LIN {X 0,Y 220.373,Z 1009.836,A -85,B 0,C 180,E1 18253.847,E2 18253.847} C_VEL
LIN {X 0,Y 219.138,Z 1016.029,A -85,B 0,C 180,E1 18268.015,E2 18268.015} C_VEL
LIN {X 0,Y 219.565,Z 1013.034,A -85,B 0,C 180,E1 18281.966,E2 18281.966} C_VEL
LIN {X 0,Y 227.617,Z 997.179,A -85,B 0,C 180,E1 18298.905,E2 18298.905} C_VEL
LIN {X 0,Y 250.356,Z 965.181,A -85,B 0,C 180,E1 18314.989,E2 18314.989} C_VEL
LIN {X 0,Y 283.389,Z 919.125,A -85,B 0,C 180,E1 18326.696,E2 18326.696} C_VEL
LIN {X 0,Y 317.274,Z 862.724,A -85,B 0,C 180,E1 18334.047,E2 18334.047} C_VEL
LIN {X 0,Y 322.512,Z 850.682,A -85,B 0,C 180,E1 18335.556,E2 18335.556} C_VEL
LIN {X 0,Y 322.481,Z 836.456,A -85,B 0,C 180,E1 18342.214,E2 18342.214} C_VEL
LIN {X 0,Y 322.225,Z 833.773,A -85,B 0,C 180,E1 18347.787,E2 18347.787} C_VEL
LIN {X 0,Y 321.726,Z 841.185,A -85,B 0,C 180,E1 18353.928,E2 18353.928} C_VEL
LIN {X 0,Y 319.566,Z 854.404,A -85,B 0,C 180,E1 18358.488,E2 18358.488} C_VEL
LIN {X 0,Y 300.592,Z 887.455,A -85,B 0,C 180,E1 18362.382,E2 18362.382} C_VEL
LIN {X 0,Y 279.885,Z 912.877,A -85,B 0,C 180,E1 18365.051,E2 18365.051} C_VEL
LIN {X 0,Y 246.942,Z 954.001,A -85,B 0,C 180,E1 18376.073,E2 18376.073} C_VEL
LIN {X 0,Y 222.563,Z 982.704,A -85,B 0,C 180,E1 18391.535,E2 18391.535} C_VEL
LIN {X 0,Y 212.303,Z 997.242,A -85,B 0,C 180,E1 18408.658,E2 18408.658} C_VEL
LIN {X 0,Y 209.744,Z 999.849,A -85,B 0,C 180,E1 18424.769,E2 18424.769} C_VEL
LIN {X 0,Y 214.305,Z 991.756,A -85,B 0,C 180,E1 18441.286,E2 18441.286} C_VEL
LIN {X 0,Y 227.941,Z 970.708,A -85,B 0,C 180,E1 18457.653,E2 18457.653} C_VEL
LIN {X 0,Y 253.573,Z 935.333,A -85,B 0,C 180,E1 18471.372,E2 18471.372} C_VEL
LIN {X 0,Y 285.146,Z 885.566,A -85,B 0,C 180,E1 18481.26,E2 18481.26} C_VEL
LIN {X 0,Y 302.468,Z 850.539,A -85,B 0,C 180,E1 18485.569,E2 18485.569} C_VEL
LIN {X 0,Y 296.04,Z 820.813,A -85,B 0,C 180,E1 18495.646,E2 18495.646} C_VEL
LIN {X 0,Y 288.186,Z 798.555,A -85,B 0,C 180,E1 18507.321,E2 18507.321} C_VEL
LIN {X 0,Y 283.718,Z 785.2,A -85,B 0,C 180,E1 18521.323,E2 18521.323} C_VEL
LIN {X 0,Y 285.026,Z 786.25,A -85,B 0,C 180,E1 18533.316,E2 18533.316} C_VEL
LIN {X 0,Y 290.912,Z 799.543,A -85,B 0,C 180,E1 18545.216,E2 18545.216} C_VEL
LIN {X 0,Y 300.284,Z 824.928,A -85,B 0,C 180,E1 18556.867,E2 18556.867} C_VEL
LIN {X 0,Y 306.026,Z 852.939,A -85,B 0,C 180,E1 18565.183,E2 18565.183} C_VEL
LIN {X 0,Y 276.942,Z 909.709,A -85,B 0,C 180,E1 18571.855,E2 18571.855} C_VEL
LIN {X 0,Y 245.558,Z 958.022,A -85,B 0,C 180,E1 18582.734,E2 18582.734} C_VEL
LIN {X 0,Y 221.833,Z 992.283,A -85,B 0,C 180,E1 18597.981,E2 18597.981} C_VEL
LIN {X 0,Y 212.147,Z 1010.601,A -85,B 0,C 180,E1 18614.772,E2 18614.772} C_VEL
LIN {X 0,Y 211.129,Z 1015.72,A -85,B 0,C 180,E1 18627.939,E2 18627.939} C_VEL
LIN {X 0,Y 211.636,Z 1012.762,A -85,B 0,C 180,E1 18642.422,E2 18642.422} C_VEL
LIN {X 0,Y 220.353,Z 997.009,A -85,B 0,C 180,E1 18659.954,E2 18659.954} C_VEL
LIN {X 0,Y 244.372,Z 965.392,A -85,B 0,C 180,E1 18676.307,E2 18676.307} C_VEL
LIN {X 0,Y 278.886,Z 919.71,A -85,B 0,C 180,E1 18688.066,E2 18688.066} C_VEL
LIN {X 0,Y 313.812,Z 864.077,A -85,B 0,C 180,E1 18695.333,E2 18695.333} C_VEL
LIN {X 0,Y 317.905,Z 855.344,A -85,B 0,C 180,E1 18696.473,E2 18696.473} C_VEL
LIN {X 0,Y 318.346,Z 842.413,A -85,B 0,C 180,E1 18703.405,E2 18703.405} C_VEL
LIN {X 0,Y 318.197,Z 842.388,A -85,B 0,C 180,E1 18710.413,E2 18710.413} C_VEL
LIN {X 0,Y 315.699,Z 857.128,A -85,B 0,C 180,E1 18717.308,E2 18717.308} C_VEL
LIN {X 0,Y 281.373,Z 910.889,A -85,B 0,C 180,E1 18724.66,E2 18724.66} C_VEL
LIN {X 0,Y 279.885,Z 912.877,A -85,B 0,C 180,E1 18725.051,E2 18725.051} C_VEL
LIN {X 0,Y 258.115,Z 935.593,A -85,B 0,C 180,E1 18728.56,E2 18728.56} C_VEL
LIN {X 0,Y 226.791,Z 970.834,A -85,B 0,C 180,E1 18742.183,E2 18742.183} C_VEL
LIN {X 0,Y 207.855,Z 992.665,A -85,B 0,C 180,E1 18759.95,E2 18759.95} C_VEL
LIN {X 0,Y 202.185,Z 999.999,A -85,B 0,C 180,E1 18775.741,E2 18775.741} C_VEL
LIN {X 0,Y 203.21,Z 997.796,A -85,B 0,C 180,E1 18792.62,E2 18792.62} C_VEL
LIN {X 0,Y 211.901,Z 983.961,A -85,B 0,C 180,E1 18809.984,E2 18809.984} C_VEL
LIN {X 0,Y 234.192,Z 954.323,A -85,B 0,C 180,E1 18826.47,E2 18826.47} C_VEL
LIN {X 0,Y 263.333,Z 913.447,A -85,B 0,C 180,E1 18837.921,E2 18837.921} C_VEL
LIN {X 0,Y 293.981,Z 860.719,A -85,B 0,C 180,E1 18845.731,E2 18845.731} C_VEL
LIN {X 0,Y 296.609,Z 852.495,A -85,B 0,C 180,E1 18847.039,E2 18847.039} C_VEL
LIN {X 0,Y 290.792,Z 824.048,A -85,B 0,C 180,E1 18857.396,E2 18857.396} C_VEL
LIN {X 0,Y 283.733,Z 803.211,A -85,B 0,C 180,E1 18869.449,E2 18869.449} C_VEL
LIN {X 0,Y 280.825,Z 792.085,A -85,B 0,C 180,E1 18882.693,E2 18882.693} C_VEL
LIN {X 0,Y 282.263,Z 794.533,A -85,B 0,C 180,E1 18894.079,E2 18894.079} C_VEL
LIN {X 0,Y 287.729,Z 807.162,A -85,B 0,C 180,E1 18905.273,E2 18905.273} C_VEL
LIN {X 0,Y 296.059,Z 832.031,A -85,B 0,C 180,E1 18916.731,E2 18916.731} C_VEL
LIN {X 0,Y 300.062,Z 857.017,A -85,B 0,C 180,E1 18924.226,E2 18924.226} C_VEL
LIN {X 0,Y 270.046,Z 912.728,A -85,B 0,C 180,E1 18931.016,E2 18931.016} C_VEL
LIN {X 0,Y 238.555,Z 959.182,A -85,B 0,C 180,E1 18941.859,E2 18941.859} C_VEL
LIN {X 0,Y 214.827,Z 991.776,A -85,B 0,C 180,E1 18956.805,E2 18956.805} C_VEL
LIN {X 0,Y 204.65,Z 1009.197,A -85,B 0,C 180,E1 18972.744,E2 18972.744} C_VEL
LIN {X 0,Y 203.132,Z 1015.411,A -85,B 0,C 180,E1 18987.858,E2 18987.858} C_VEL
LIN {X 0,Y 203.701,Z 1012.495,A -85,B 0,C 180,E1 19002.914,E2 19002.914} C_VEL
LIN {X 0,Y 213.159,Z 996.874,A -85,B 0,C 180,E1 19021.055,E2 19021.055} C_VEL
LIN {X 0,Y 239.014,Z 965.037,A -85,B 0,C 180,E1 19037.919,E2 19037.919} C_VEL
LIN {X 0,Y 275.385,Z 919.278,A -85,B 0,C 180,E1 19049.672,E2 19049.672} C_VEL
LIN {X 0,Y 311.753,Z 863.373,A -85,B 0,C 180,E1 19056.851,E2 19056.851} C_VEL
LIN {X 0,Y 313.841,Z 854.831,A -85,B 0,C 180,E1 19059.622,E2 19059.622} C_VEL
LIN {X 0,Y 314.074,Z 848.409,A -85,B 0,C 180,E1 19064.613,E2 19064.613} C_VEL
LIN {X 0,Y 313.639,Z 850.576,A -85,B 0,C 180,E1 19071.382,E2 19071.382} C_VEL
LIN {X 0,Y 310.047,Z 863.365,A -85,B 0,C 180,E1 19076.454,E2 19076.454} C_VEL
LIN {X 0,Y 273.828,Z 916.35,A -85,B 0,C 180,E1 19084.114,E2 19084.114} C_VEL
LIN {X 0,Y 258.115,Z 935.593,A -85,B 0,C 180,E1 19088.56,E2 19088.56} C_VEL
LIN {X 0,Y 236.075,Z 955.304,A -85,B 0,C 180,E1 19093.128,E2 19093.128} C_VEL
LIN {X 0,Y 208.191,Z 984.166,A -85,B 0,C 180,E1 19109.592,E2 19109.592} C_VEL
LIN {X 0,Y 196.123,Z 998.481,A -85,B 0,C 180,E1 19128.875,E2 19128.875} C_VEL
LIN {X 0,Y 193.672,Z 1000.479,A -85,B 0,C 180,E1 19144.472,E2 19144.472} C_VEL
LIN {X 0,Y 197.918,Z 993.812,A -85,B 0,C 180,E1 19160.495,E2 19160.495} C_VEL
LIN {X 0,Y 211.983,Z 974.227,A -85,B 0,C 180,E1 19178.233,E2 19178.233} C_VEL
LIN {X 0,Y 239.645,Z 939.396,A -85,B 0,C 180,E1 19193.058,E2 19193.058} C_VEL
LIN {X 0,Y 272.06,Z 892.564,A -85,B 0,C 180,E1 19203.038,E2 19203.038} C_VEL
LIN {X 0,Y 291.019,Z 856.591,A -85,B 0,C 180,E1 19207.905,E2 19207.905} C_VEL
LIN {X 0,Y 285.972,Z 828.948,A -85,B 0,C 180,E1 19218.435,E2 19218.435} C_VEL
LIN {X 0,Y 280.548,Z 811.013,A -85,B 0,C 180,E1 19229.064,E2 19229.064} C_VEL
LIN {X 0,Y 277.851,Z 799.48,A -85,B 0,C 180,E1 19242.909,E2 19242.909} C_VEL
LIN {X 0,Y 279.25,Z 801.961,A -85,B 0,C 180,E1 19254.015,E2 19254.015} C_VEL
LIN {X 0,Y 284.31,Z 814.699,A -85,B 0,C 180,E1 19265.337,E2 19265.337} C_VEL
LIN {X 0,Y 291.619,Z 838.957,A -85,B 0,C 180,E1 19276.605,E2 19276.605} C_VEL
LIN {X 0,Y 294.508,Z 860.273,A -85,B 0,C 180,E1 19283.162,E2 19283.162} C_VEL
LIN {X 0,Y 263.242,Z 915.713,A -85,B 0,C 180,E1 19290.144,E2 19290.144} C_VEL
LIN {X 0,Y 231.356,Z 960.576,A -85,B 0,C 180,E1 19301.03,E2 19301.03} C_VEL
LIN {X 0,Y 206.727,Z 992.867,A -85,B 0,C 180,E1 19316.592,E2 19316.592} C_VEL
LIN {X 0,Y 196.236,Z 1010.295,A -85,B 0,C 180,E1 19334.295,E2 19334.295} C_VEL
LIN {X 0,Y 195.12,Z 1015.1,A -85,B 0,C 180,E1 19347.77,E2 19347.77} C_VEL
LIN {X 0,Y 195.48,Z 1013.18,A -85,B 0,C 180,E1 19361.19,E2 19361.19} C_VEL
LIN {X 0,Y 204.534,Z 998.649,A -85,B 0,C 180,E1 19380.621,E2 19380.621} C_VEL
LIN {X 0,Y 230.077,Z 968.974,A -85,B 0,C 180,E1 19397.905,E2 19397.905} C_VEL
LIN {X 0,Y 266.944,Z 925.543,A -85,B 0,C 180,E1 19410.107,E2 19410.107} C_VEL
LIN {X 0,Y 306.085,Z 869.504,A -85,B 0,C 180,E1 19417.76,E2 19417.76} C_VEL
LIN {X 0,Y 309.026,Z 862.483,A -85,B 0,C 180,E1 19419.29,E2 19419.29} C_VEL
LIN {X 0,Y 309.799,Z 855.412,A -85,B 0,C 180,E1 19424.396,E2 19424.396} C_VEL
LIN {X 0,Y 309.551,Z 855.889,A -85,B 0,C 180,E1 19430.143,E2 19430.143} C_VEL
LIN {X 0,Y 306.388,Z 866.253,A -85,B 0,C 180,E1 19435.226,E2 19435.226} C_VEL
LIN {X 0,Y 268.378,Z 919.194,A -85,B 0,C 180,E1 19442.994,E2 19442.994} C_VEL
LIN {X 0,Y 236.075,Z 955.304,A -85,B 0,C 180,E1 19453.128,E2 19453.128} C_VEL
LIN {X 0,Y 214.987,Z 971.635,A -85,B 0,C 180,E1 19459.091,E2 19459.091} C_VEL
LIN {X 0,Y 192.996,Z 993.395,A -85,B 0,C 180,E1 19477.924,E2 19477.924} C_VEL
LIN {X 0,Y 186.819,Z 1000.134,A -85,B 0,C 180,E1 19492.466,E2 19492.466} C_VEL
LIN {X 0,Y 186.364,Z 999.741,A -85,B 0,C 180,E1 19509.501,E2 19509.501} C_VEL
LIN {X 0,Y 192.215,Z 990.787,A -85,B 0,C 180,E1 19525.532,E2 19525.532} C_VEL
LIN {X 0,Y 211.117,Z 967.464,A -85,B 0,C 180,E1 19543.533,E2 19543.533} C_VEL
LIN {X 0,Y 242.514,Z 928.84,A -85,B 0,C 180,E1 19557.485,E2 19557.485} C_VEL
LIN {X 0,Y 276.181,Z 878.662,A -85,B 0,C 180,E1 19566.452,E2 19566.452} C_VEL
LIN {X 0,Y 285.512,Z 860.953,A -85,B 0,C 180,E1 19568.708,E2 19568.708} C_VEL
LIN {X 0,Y 281.244,Z 834.112,A -85,B 0,C 180,E1 19579.384,E2 19579.384} C_VEL
LIN {X 0,Y 276.401,Z 816.717,A -85,B 0,C 180,E1 19590.458,E2 19590.458} C_VEL
LIN {X 0,Y 274.593,Z 806.641,A -85,B 0,C 180,E1 19605.281,E2 19605.281} C_VEL
LIN {X 0,Y 276.326,Z 810.262,A -85,B 0,C 180,E1 19615.255,E2 19615.255} C_VEL
LIN {X 0,Y 281.536,Z 824.755,A -85,B 0,C 180,E1 19626.942,E2 19626.942} C_VEL
LIN {X 0,Y 287.874,Z 850.107,A -85,B 0,C 180,E1 19638.014,E2 19638.014} C_VEL
LIN {X 0,Y 288.564,Z 864.213,A -85,B 0,C 180,E1 19642.155,E2 19642.155} C_VEL
LIN {X 0,Y 256.518,Z 918.691,A -85,B 0,C 180,E1 19649.236,E2 19649.236} C_VEL
LIN {X 0,Y 222.348,Z 964.299,A -85,B 0,C 180,E1 19660.992,E2 19660.992} C_VEL
LIN {X 0,Y 197.99,Z 994.596,A -85,B 0,C 180,E1 19676.98,E2 19676.98} C_VEL
LIN {X 0,Y 188.368,Z 1009.917,A -85,B 0,C 180,E1 19693.621,E2 19693.621} C_VEL
LIN {X 0,Y 187.121,Z 1014.79,A -85,B 0,C 180,E1 19707.675,E2 19707.675} C_VEL
LIN {X 0,Y 187.765,Z 1012.235,A -85,B 0,C 180,E1 19723.373,E2 19723.373} C_VEL
LIN {X 0,Y 198.68,Z 997.07,A -85,B 0,C 180,E1 19743.168,E2 19743.168} C_VEL
LIN {X 0,Y 228.668,Z 964.789,A -85,B 0,C 180,E1 19761.194,E2 19761.194} C_VEL
LIN {X 0,Y 268.282,Z 919.662,A -85,B 0,C 180,E1 19772.816,E2 19772.816} C_VEL
LIN {X 0,Y 304.265,Z 868.851,A -85,B 0,C 180,E1 19779.581,E2 19779.581} C_VEL
LIN {X 0,Y 305.188,Z 861.542,A -85,B 0,C 180,E1 19785.849,E2 19785.849} C_VEL
LIN {X 0,Y 304.29,Z 864.506,A -85,B 0,C 180,E1 19791.418,E2 19791.418} C_VEL
LIN {X 0,Y 300.81,Z 872.287,A -85,B 0,C 180,E1 19794.309,E2 19794.309} C_VEL
LIN {X 0,Y 261.63,Z 923.52,A -85,B 0,C 180,E1 19802.173,E2 19802.173} C_VEL
LIN {X 0,Y 224.173,Z 962.683,A -85,B 0,C 180,E1 19814.39,E2 19814.39} C_VEL
LIN {X 0,Y 214.987,Z 971.635,A -85,B 0,C 180,E1 19819.091,E2 19819.091} C_VEL
LIN {X 0,Y 195.178,Z 984.685,A -85,B 0,C 180,E1 19826.484,E2 19826.484} C_VEL
LIN {X 0,Y 181.146,Z 998.421,A -85,B 0,C 180,E1 19845.432,E2 19845.432} C_VEL
LIN {X 0,Y 177.585,Z 1001.129,A -85,B 0,C 180,E1 19863.839,E2 19863.839} C_VEL
LIN {X 0,Y 181.808,Z 995.317,A -85,B 0,C 180,E1 19880.391,E2 19880.391} C_VEL
LIN {X 0,Y 197.338,Z 975.911,A -85,B 0,C 180,E1 19899.965,E2 19899.965} C_VEL
LIN {X 0,Y 226.305,Z 942.826,A -85,B 0,C 180,E1 19915.118,E2 19915.118} C_VEL
LIN {X 0,Y 261.524,Z 895.866,A -85,B 0,C 180,E1 19925.53,E2 19925.53} C_VEL
LIN {X 0,Y 279.861,Z 863.813,A -85,B 0,C 180,E1 19930.039,E2 19930.039} C_VEL
LIN {X 0,Y 276.366,Z 838.353,A -85,B 0,C 180,E1 19940.829,E2 19940.829} C_VEL
LIN {X 0,Y 272.298,Z 822.591,A -85,B 0,C 180,E1 19951.71,E2 19951.71} C_VEL
LIN {X 0,Y 271.325,Z 813.923,A -85,B 0,C 180,E1 19965.405,E2 19965.405} C_VEL
LIN {X 0,Y 272.968,Z 817.502,A -85,B 0,C 180,E1 19975.196,E2 19975.196} C_VEL
LIN {X 0,Y 277.749,Z 832.214,A -85,B 0,C 180,E1 19987.038,E2 19987.038} C_VEL
LIN {X 0,Y 283.068,Z 857.304,A -85,B 0,C 180,E1 19998.07,E2 19998.07} C_VEL
LIN {X 0,Y 282.572,Z 868.253,A -85,B 0,C 180,E1 20001.117,E2 20001.117} C_VEL
LIN {X 0,Y 249.814,Z 921.374,A -85,B 0,C 180,E1 20008.253,E2 20008.253} C_VEL
LIN {X 0,Y 215.743,Z 964.986,A -85,B 0,C 180,E1 20019.832,E2 20019.832} C_VEL
LIN {X 0,Y 189.597,Z 995.901,A -85,B 0,C 180,E1 20037.098,E2 20037.098} C_VEL
LIN {X 0,Y 179.879,Z 1011.008,A -85,B 0,C 180,E1 20055.766,E2 20055.766} C_VEL
LIN {X 0,Y 179.299,Z 1014.62,A -85,B 0,C 180,E1 20072.424,E2 20072.424} C_VEL
LIN {X 0,Y 182.377,Z 1007.844,A -85,B 0,C 180,E1 20091.989,E2 20091.989} C_VEL
LIN {X 0,Y 201.967,Z 986.21,A -85,B 0,C 180,E1 20112.551,E2 20112.551} C_VEL
LIN {X 0,Y 238.666,Z 949.421,A -85,B 0,C 180,E1 20127.929,E2 20127.929} C_VEL
LIN {X 0,Y 280.238,Z 901.075,A -85,B 0,C 180,E1 20137.335,E2 20137.335} C_VEL
LIN {X 0,Y 299.708,Z 873.201,A -85,B 0,C 180,E1 20140.812,E2 20140.812} C_VEL
LIN {X 0,Y 300.756,Z 867.825,A -85,B 0,C 180,E1 20146.901,E2 20146.901} C_VEL
LIN {X 0,Y 298.717,Z 872.659,A -85,B 0,C 180,E1 20152.131,E2 20152.131} C_VEL
LIN {X 0,Y 293.823,Z 880.361,A -85,B 0,C 180,E1 20153.608,E2 20153.608} C_VEL
LIN {X 0,Y 253.158,Z 929.782,A -85,B 0,C 180,E1 20161.74,E2 20161.74} C_VEL
LIN {X 0,Y 214.089,Z 967.716,A -85,B 0,C 180,E1 20174.957,E2 20174.957} C_VEL
LIN {X 0,Y 195.178,Z 984.685,A -85,B 0,C 180,E1 20186.484,E2 20186.484} C_VEL
LIN {X 0,Y 178.309,Z 994.199,A -85,B 0,C 180,E1 20195.666,E2 20195.666} C_VEL
LIN {X 0,Y 170.224,Z 1001.371,A -85,B 0,C 180,E1 20214.587,E2 20214.587} C_VEL
LIN {X 0,Y 171.766,Z 998.594,A -85,B 0,C 180,E1 20235.07,E2 20235.07} C_VEL
LIN {X 0,Y 183.906,Z 983.75,A -85,B 0,C 180,E1 20255.332,E2 20255.332} C_VEL
LIN {X 0,Y 211.438,Z 954.189,A -85,B 0,C 180,E1 20272.694,E2 20272.694} C_VEL
LIN {X 0,Y 247.11,Z 910.522,A -85,B 0,C 180,E1 20284.617,E2 20284.617} C_VEL
LIN {X 0,Y 274.285,Z 868.117,A -85,B 0,C 180,E1 20290.87,E2 20290.87} C_VEL
LIN {X 0,Y 271.715,Z 844.511,A -85,B 0,C 180,E1 20301.256,E2 20301.256} C_VEL
LIN {X 0,Y 268.173,Z 827.819,A -85,B 0,C 180,E1 20313.613,E2 20313.613} C_VEL
LIN {X 0,Y 267.755,Z 821.155,A -85,B 0,C 180,E1 20325.206,E2 20325.206} C_VEL
LIN {X 0,Y 269.313,Z 824.6,A -85,B 0,C 180,E1 20335.131,E2 20335.131} C_VEL
LIN {X 0,Y 273.617,Z 839.556,A -85,B 0,C 180,E1 20347.144,E2 20347.144} C_VEL
LIN {X 0,Y 277.981,Z 863.95,A -85,B 0,C 180,E1 20357.976,E2 20357.976} C_VEL
LIN {X 0,Y 277.354,Z 870.945,A -85,B 0,C 180,E1 20359.909,E2 20359.909} C_VEL
LIN {X 0,Y 242.904,Z 924.412,A -85,B 0,C 180,E1 20367.306,E2 20367.306} C_VEL
LIN {X 0,Y 208.121,Z 966.819,A -85,B 0,C 180,E1 20379.087,E2 20379.087} C_VEL
LIN {X 0,Y 181.35,Z 996.976,A -85,B 0,C 180,E1 20397.047,E2 20397.047} C_VEL
LIN {X 0,Y 171.656,Z 1011.578,A -85,B 0,C 180,E1 20417.23,E2 20417.23} C_VEL
LIN {X 0,Y 171.299,Z 1014.33,A -85,B 0,C 180,E1 20432.538,E2 20432.538} C_VEL
LIN {X 0,Y 174.747,Z 1007.653,A -85,B 0,C 180,E1 20453.003,E2 20453.003} C_VEL
LIN {X 0,Y 195.931,Z 986.211,A -85,B 0,C 180,E1 20474.193,E2 20474.193} C_VEL
LIN {X 0,Y 234.661,Z 949.6,A -85,B 0,C 180,E1 20489.701,E2 20489.701} C_VEL
LIN {X 0,Y 277.708,Z 901.724,A -85,B 0,C 180,E1 20498.913,E2 20498.913} C_VEL
LIN {X 0,Y 295.194,Z 877.852,A -85,B 0,C 180,E1 20502.003,E2 20502.003} C_VEL
LIN {X 0,Y 295.893,Z 874.332,A -85,B 0,C 180,E1 20506.681,E2 20506.681} C_VEL
LIN {X 0,Y 294.382,Z 877.613,A -85,B 0,C 180,E1 20511.127,E2 20511.127} C_VEL
LIN {X 0,Y 285.888,Z 889.367,A -85,B 0,C 180,E1 20513.015,E2 20513.015} C_VEL
LIN {X 0,Y 242.563,Z 937.712,A -85,B 0,C 180,E1 20521.816,E2 20521.816} C_VEL
LIN {X 0,Y 203.626,Z 972.739,A -85,B 0,C 180,E1 20535.745,E2 20535.745} C_VEL
LIN {X 0,Y 178.309,Z 994.199,A -85,B 0,C 180,E1 20555.666,E2 20555.666} C_VEL
LIN {X 0,Y 164.556,Z 1000.038,A -85,B 0,C 180,E1 20566.474,E2 20566.474} C_VEL
LIN {X 0,Y 161.52,Z 1001.635,A -85,B 0,C 180,E1 20584.989,E2 20584.989} C_VEL
LIN {X 0,Y 167.196,Z 994.523,A -85,B 0,C 180,E1 20604.065,E2 20604.065} C_VEL
LIN {X 0,Y 185.998,Z 974.459,A -85,B 0,C 180,E1 20624.17,E2 20624.17} C_VEL
LIN {X 0,Y 219.864,Z 938.759,A -85,B 0,C 180,E1 20639.736,E2 20639.736} C_VEL
LIN {X 0,Y 256.908,Z 890.924,A -85,B 0,C 180,E1 20649.422,E2 20649.422} C_VEL
LIN {X 0,Y 268.754,Z 871.501,A -85,B 0,C 180,E1 20652.088,E2 20652.088} C_VEL
LIN {X 0,Y 266.547,Z 848.04,A -85,B 0,C 180,E1 20663.274,E2 20663.274} C_VEL
LIN {X 0,Y 263.872,Z 833.458,A -85,B 0,C 180,E1 20675.405,E2 20675.405} C_VEL
LIN {X 0,Y 264.119,Z 828.357,A -85,B 0,C 180,E1 20684.997,E2 20684.997} C_VEL
LIN {X 0,Y 265.597,Z 831.676,A -85,B 0,C 180,E1 20695.063,E2 20695.063} C_VEL
LIN {X 0,Y 269.418,Z 846.849,A -85,B 0,C 180,E1 20707.256,E2 20707.256} C_VEL
LIN {X 0,Y 272.863,Z 872.154,A -85,B 0,C 180,E1 20718.45,E2 20718.45} C_VEL
LIN {X 0,Y 236.605,Z 926.633,A -85,B 0,C 180,E1 20726.149,E2 20726.149} C_VEL
LIN {X 0,Y 200.551,Z 968.529,A -85,B 0,C 180,E1 20738.271,E2 20738.271} C_VEL
LIN {X 0,Y 174.22,Z 996.662,A -85,B 0,C 180,E1 20755.754,E2 20755.754} C_VEL
LIN {X 0,Y 163.747,Z 1011.207,A -85,B 0,C 180,E1 20776.602,E2 20776.602} C_VEL
LIN {X 0,Y 163.273,Z 1014.039,A -85,B 0,C 180,E1 20792.663,E2 20792.663} C_VEL
LIN {X 0,Y 167.187,Z 1007.471,A -85,B 0,C 180,E1 20814.108,E2 20814.108} C_VEL
LIN {X 0,Y 190.062,Z 986.24,A -85,B 0,C 180,E1 20835.94,E2 20835.94} C_VEL
LIN {X 0,Y 230.967,Z 949.773,A -85,B 0,C 180,E1 20851.549,E2 20851.549} C_VEL
LIN {X 0,Y 275.608,Z 902.207,A -85,B 0,C 180,E1 20860.563,E2 20860.563} C_VEL
LIN {X 0,Y 290.368,Z 883.179,A -85,B 0,C 180,E1 20862.929,E2 20862.929} C_VEL
LIN {X 0,Y 290.418,Z 881.739,A -85,B 0,C 180,E1 20869.486,E2 20869.486} C_VEL
LIN {X 0,Y 287.671,Z 885.69,A -85,B 0,C 180,E1 20870.88,E2 20870.88} C_VEL
LIN {X 0,Y 244.957,Z 932.993,A -85,B 0,C 180,E1 20878.66,E2 20878.66} C_VEL
LIN {X 0,Y 202.336,Z 970.133,A -85,B 0,C 180,E1 20891.992,E2 20891.992} C_VEL
LIN {X 0,Y 172.136,Z 993.852,A -85,B 0,C 180,E1 20913.12,E2 20913.12} C_VEL
LIN {X 0,Y 164.556,Z 1000.038,A -85,B 0,C 180,E1 20926.474,E2 20926.474} C_VEL
LIN {X 0,Y 153.429,Z 1002.188,A -85,B 0,C 180,E1 20938.59,E2 20938.59} C_VEL
LIN {X 0,Y 157.012,Z 997.935,A -85,B 0,C 180,E1 20958.855,E2 20958.855} C_VEL
LIN {X 0,Y 173.577,Z 980.588,A -85,B 0,C 180,E1 20981.346,E2 20981.346} C_VEL
LIN {X 0,Y 206.537,Z 948.078,A -85,B 0,C 180,E1 20998.53,E2 20998.53} C_VEL
LIN {X 0,Y 244.476,Z 903.259,A -85,B 0,C 180,E1 21009.193,E2 21009.193} C_VEL
LIN {X 0,Y 263.207,Z 874.609,A -85,B 0,C 180,E1 21013.495,E2 21013.495} C_VEL
LIN {X 0,Y 261.721,Z 852.87,A -85,B 0,C 180,E1 21024.553,E2 21024.553} C_VEL
LIN {X 0,Y 260.003,Z 840.909,A -85,B 0,C 180,E1 21034.785,E2 21034.785} C_VEL
LIN {X 0,Y 260.189,Z 835.421,A -85,B 0,C 180,E1 21044.765,E2 21044.765} C_VEL
LIN {X 0,Y 261.613,Z 838.627,A -85,B 0,C 180,E1 21054.987,E2 21054.987} C_VEL
LIN {X 0,Y 264.696,Z 852.603,A -85,B 0,C 180,E1 21066.56,E2 21066.56} C_VEL
LIN {X 0,Y 267.282,Z 875.661,A -85,B 0,C 180,E1 21077.292,E2 21077.292} C_VEL
LIN {X 0,Y 230.2,Z 929.08,A -85,B 0,C 180,E1 21084.981,E2 21084.981} C_VEL
LIN {X 0,Y 191.019,Z 972.326,A -85,B 0,C 180,E1 21098.32,E2 21098.32} C_VEL
LIN {X 0,Y 163.969,Z 999.775,A -85,B 0,C 180,E1 21118.007,E2 21118.007} C_VEL
LIN {X 0,Y 155.852,Z 1010.834,A -85,B 0,C 180,E1 21135.909,E2 21135.909} C_VEL
LIN {X 0,Y 155.244,Z 1013.749,A -85,B 0,C 180,E1 21152.8,E2 21152.8} C_VEL
LIN {X 0,Y 158.379,Z 1008.67,A -85,B 0,C 180,E1 21172.536,E2 21172.536} C_VEL
LIN {X 0,Y 180.514,Z 989.415,A -85,B 0,C 180,E1 21195.609,E2 21195.609} C_VEL
LIN {X 0,Y 222.911,Z 954.247,A -85,B 0,C 180,E1 21212.256,E2 21212.256} C_VEL
LIN {X 0,Y 269.734,Z 907.369,A -85,B 0,C 180,E1 21221.63,E2 21221.63} C_VEL
LIN {X 0,Y 285.448,Z 888.358,A -85,B 0,C 180,E1 21224.119,E2 21224.119} C_VEL
LIN {X 0,Y 284.666,Z 888.74,A -85,B 0,C 180,E1 21229.512,E2 21229.512} C_VEL
LIN {X 0,Y 240.036,Z 935.681,A -85,B 0,C 180,E1 21237.289,E2 21237.289} C_VEL
LIN {X 0,Y 197.13,Z 971.013,A -85,B 0,C 180,E1 21250.188,E2 21250.188} C_VEL
LIN {X 0,Y 166.462,Z 993.26,A -85,B 0,C 180,E1 21270.123,E2 21270.123} C_VEL
LIN {X 0,Y 155.022,Z 1001.541,A -85,B 0,C 180,E1 21290.484,E2 21290.484} C_VEL
LIN {X 0,Y 153.429,Z 1002.188,A -85,B 0,C 180,E1 21298.59,E2 21298.59} C_VEL
LIN {X 0,Y 146.468,Z 1000.724,A -85,B 0,C 180,E1 21311.913,E2 21311.913} C_VEL
LIN {X 0,Y 156.5,Z 990.564,A -85,B 0,C 180,E1 21332.78,E2 21332.78} C_VEL
LIN {X 0,Y 183.911,Z 965.333,A -85,B 0,C 180,E1 21353.077,E2 21353.077} C_VEL
LIN {X 0,Y 221.175,Z 927.29,A -85,B 0,C 180,E1 21366.286,E2 21366.286} C_VEL
LIN {X 0,Y 257.636,Z 878.857,A -85,B 0,C 180,E1 21374.432,E2 21374.432} C_VEL
LIN {X 0,Y 256.803,Z 857.712,A -85,B 0,C 180,E1 21385.833,E2 21385.833} C_VEL
LIN {X 0,Y 255.488,Z 846.13,A -85,B 0,C 180,E1 21397.272,E2 21397.272} C_VEL
LIN {X 0,Y 256.7,Z 842.254,A -85,B 0,C 180,E1 21408.039,E2 21408.039} C_VEL
LIN {X 0,Y 258.539,Z 850.238,A -85,B 0,C 180,E1 21419.977,E2 21419.977} C_VEL
LIN {X 0,Y 261.205,Z 869.219,A -85,B 0,C 180,E1 21431.705,E2 21431.705} C_VEL
LIN {X 0,Y 260.859,Z 880.744,A -85,B 0,C 180,E1 21436.275,E2 21436.275} C_VEL
LIN {X 0,Y 223.843,Z 931.314,A -85,B 0,C 180,E1 21443.755,E2 21443.755} C_VEL
LIN {X 0,Y 184.776,Z 972.627,A -85,B 0,C 180,E1 21456.794,E2 21456.794} C_VEL
LIN {X 0,Y 157.366,Z 998.811,A -85,B 0,C 180,E1 21475.898,E2 21475.898} C_VEL
LIN {X 0,Y 147.47,Z 1011.178,A -85,B 0,C 180,E1 21497.575,E2 21497.575} C_VEL
LIN {X 0,Y 147.214,Z 1013.461,A -85,B 0,C 180,E1 21512.953,E2 21512.953} C_VEL
LIN {X 0,Y 150.801,Z 1008.473,A -85,B 0,C 180,E1 21533.736,E2 21533.736} C_VEL
LIN {X 0,Y 174.793,Z 989.497,A -85,B 0,C 180,E1 21557.559,E2 21557.559} C_VEL
LIN {X 0,Y 220.666,Z 953.584,A -85,B 0,C 180,E1 21574.507,E2 21574.507} C_VEL
LIN {X 0,Y 270.024,Z 905.815,A -85,B 0,C 180,E1 21583.612,E2 21583.612} C_VEL
LIN {X 0,Y 280.391,Z 893.865,A -85,B 0,C 180,E1 21585.13,E2 21585.13} C_VEL
LIN {X 0,Y 279.209,Z 894.767,A -85,B 0,C 180,E1 21588.464,E2 21588.464} C_VEL
LIN {X 0,Y 231.031,Z 942.062,A -85,B 0,C 180,E1 21596.78,E2 21596.78} C_VEL
LIN {X 0,Y 186.039,Z 976.161,A -85,B 0,C 180,E1 21610.965,E2 21610.965} C_VEL
LIN {X 0,Y 155.136,Z 996.741,A -85,B 0,C 180,E1 21633.75,E2 21633.75} C_VEL
LIN {X 0,Y 145.863,Z 1002.487,A -85,B 0,C 180,E1 21655.096,E2 21655.096} C_VEL
LIN {X 0,Y 146.468,Z 1000.724,A -85,B 0,C 180,E1 21671.913,E2 21671.913} C_VEL
LIN {X 0,Y 143.749,Z 995.928,A -85,B 0,C 180,E1 21685.876,E2 21685.876} C_VEL
LIN {X 0,Y 166.272,Z 976.023,A -85,B 0,C 180,E1 21708.631,E2 21708.631} C_VEL
LIN {X 0,Y 203.989,Z 941.181,A -85,B 0,C 180,E1 21724.561,E2 21724.561} C_VEL
LIN {X 0,Y 244.091,Z 894.263,A -85,B 0,C 180,E1 21733.997,E2 21733.997} C_VEL
LIN {X 0,Y 252.142,Z 881.384,A -85,B 0,C 180,E1 21736.186,E2 21736.186} C_VEL
LIN {X 0,Y 251.938,Z 862.573,A -85,B 0,C 180,E1 21747.156,E2 21747.156} C_VEL
LIN {X 0,Y 251.423,Z 850.919,A -85,B 0,C 180,E1 21760.593,E2 21760.593} C_VEL
LIN {X 0,Y 253.052,Z 850.036,A -85,B 0,C 180,E1 21771.707,E2 21771.707} C_VEL
LIN {X 0,Y 254.896,Z 862.628,A -85,B 0,C 180,E1 21784.243,E2 21784.243} C_VEL
LIN {X 0,Y 255.917,Z 883.314,A -85,B 0,C 180,E1 21794.902,E2 21794.902} C_VEL
LIN {X 0,Y 216.451,Z 934.858,A -85,B 0,C 180,E1 21802.745,E2 21802.745} C_VEL
LIN {X 0,Y 177.507,Z 973.914,A -85,B 0,C 180,E1 21815.687,E2 21815.687} C_VEL
LIN {X 0,Y 148.985,Z 999.775,A -85,B 0,C 180,E1 21835.926,E2 21835.926} C_VEL
LIN {X 0,Y 139.163,Z 1011.838,A -85,B 0,C 180,E1 21860.584,E2 21860.584} C_VEL
LIN {X 0,Y 139.171,Z 1012.674,A -85,B 0,C 180,E1 21879.413,E2 21879.413} C_VEL
LIN {X 0,Y 151.079,Z 1002.351,A -85,B 0,C 180,E1 21905.929,E2 21905.929} C_VEL
LIN {X 0,Y 188.064,Z 976.451,A -85,B 0,C 180,E1 21927.917,E2 21927.917} C_VEL
LIN {X 0,Y 239.81,Z 934.929,A -85,B 0,C 180,E1 21941.014,E2 21941.014} C_VEL
LIN {X 0,Y 275.099,Z 899.416,A -85,B 0,C 180,E1 21946.278,E2 21946.278} C_VEL
LIN {X 0,Y 271.883,Z 902.842,A -85,B 0,C 180,E1 21947.634,E2 21947.634} C_VEL
LIN {X 0,Y 220.443,Z 949.297,A -85,B 0,C 180,E1 21956.566,E2 21956.566} C_VEL
LIN {X 0,Y 173.105,Z 982.02,A -85,B 0,C 180,E1 21972.691,E2 21972.691} C_VEL
LIN {X 0,Y 144.198,Z 999.526,A -85,B 0,C 180,E1 21997.879,E2 21997.879} C_VEL
LIN {X 0,Y 137.26,Z 1002.857,A -85,B 0,C 180,E1 22020.164,E2 22020.164} C_VEL
LIN {X 0,Y 142.867,Z 996.953,A -85,B 0,C 180,E1 22043.904,E2 22043.904} C_VEL
LIN {X 0,Y 143.749,Z 995.928,A -85,B 0,C 180,E1 22045.876,E2 22045.876} C_VEL
LIN {X 0,Y 145.962,Z 987.941,A -85,B 0,C 180,E1 22059.576,E2 22059.576} C_VEL
LIN {X 0,Y 179.916,Z 959.886,A -85,B 0,C 180,E1 22079.708,E2 22079.708} C_VEL
LIN {X 0,Y 221.487,Z 918.333,A -85,B 0,C 180,E1 22091.918,E2 22091.918} C_VEL
LIN {X 0,Y 246.63,Z 886.275,A -85,B 0,C 180,E1 22096.896,E2 22096.896} C_VEL
LIN {X 0,Y 247.044,Z 867.49,A -85,B 0,C 180,E1 22108.508,E2 22108.508} C_VEL
LIN {X 0,Y 247.2,Z 857.067,A -85,B 0,C 180,E1 22122.097,E2 22122.097} C_VEL
LIN {X 0,Y 248.777,Z 856.508,A -85,B 0,C 180,E1 22131.207,E2 22131.207} C_VEL
LIN {X 0,Y 250.032,Z 868.214,A -85,B 0,C 180,E1 22143.455,E2 22143.455} C_VEL
LIN {X 0,Y 250.455,Z 886.592,A -85,B 0,C 180,E1 22153.566,E2 22153.566} C_VEL
LIN {X 0,Y 209.347,Z 938.027,A -85,B 0,C 180,E1 22161.589,E2 22161.589} C_VEL
LIN {X 0,Y 166.776,Z 978.335,A -85,B 0,C 180,E1 22176.203,E2 22176.203} C_VEL
LIN {X 0,Y 138.73,Z 1002.487,A -85,B 0,C 180,E1 22198.692,E2 22198.692} C_VEL
LIN {X 0,Y 131.181,Z 1011.445,A -85,B 0,C 180,E1 22220.005,E2 22220.005} C_VEL
LIN {X 0,Y 131.187,Z 1012.388,A -85,B 0,C 180,E1 22239.991,E2 22239.991} C_VEL
LIN {X 0,Y 142.5,Z 1003.568,A -85,B 0,C 180,E1 22265.854,E2 22265.854} C_VEL
LIN {X 0,Y 181.169,Z 978.474,A -85,B 0,C 180,E1 22289.158,E2 22289.158} C_VEL
LIN {X 0,Y 232.888,Z 939.651,A -85,B 0,C 180,E1 22302.124,E2 22302.124} C_VEL
LIN {X 0,Y 264.457,Z 910.464,A -85,B 0,C 180,E1 22306.75,E2 22306.75} C_VEL
LIN {X 0,Y 214.195,Z 952.798,A -85,B 0,C 180,E1 22315.314,E2 22315.314} C_VEL
LIN {X 0,Y 167.146,Z 983.279,A -85,B 0,C 180,E1 22330.938,E2 22330.938} C_VEL
LIN {X 0,Y 138.075,Z 999.299,A -85,B 0,C 180,E1 22354.482,E2 22354.482} C_VEL
LIN {X 0,Y 129.383,Z 1003.262,A -85,B 0,C 180,E1 22378.143,E2 22378.143} C_VEL
LIN {X 0,Y 134.556,Z 997.835,A -85,B 0,C 180,E1 22403.525,E2 22403.525} C_VEL
LIN {X 0,Y 145.962,Z 987.941,A -85,B 0,C 180,E1 22419.576,E2 22419.576} C_VEL
LIN {X 0,Y 153.689,Z 976.993,A -85,B 0,C 180,E1 22432.189,E2 22432.189} C_VEL
LIN {X 0,Y 193.918,Z 942.999,A -85,B 0,C 180,E1 22448.098,E2 22448.098} C_VEL
LIN {X 0,Y 235.984,Z 896.89,A -85,B 0,C 180,E1 22457.224,E2 22457.224} C_VEL
LIN {X 0,Y 241.208,Z 889.137,A -85,B 0,C 180,E1 22458.638,E2 22458.638} C_VEL
LIN {X 0,Y 242.075,Z 872.73,A -85,B 0,C 180,E1 22469.566,E2 22469.566} C_VEL
LIN {X 0,Y 242.93,Z 863.102,A -85,B 0,C 180,E1 22483.654,E2 22483.654} C_VEL
LIN {X 0,Y 244.149,Z 864.335,A -85,B 0,C 180,E1 22492.837,E2 22492.837} C_VEL
LIN {X 0,Y 245.143,Z 876.113,A -85,B 0,C 180,E1 22504.412,E2 22504.412} C_VEL
LIN {X 0,Y 244.271,Z 890.976,A -85,B 0,C 180,E1 22512.302,E2 22512.302} C_VEL
LIN {X 0,Y 202.342,Z 940.925,A -85,B 0,C 180,E1 22520.359,E2 22520.359} C_VEL
LIN {X 0,Y 160.182,Z 978.969,A -85,B 0,C 180,E1 22534.64,E2 22534.64} C_VEL
LIN {X 0,Y 130.587,Z 1002.967,A -85,B 0,C 180,E1 22558.467,E2 22558.467} C_VEL
LIN {X 0,Y 123.23,Z 1011.047,A -85,B 0,C 180,E1 22579.353,E2 22579.353} C_VEL
LIN {X 0,Y 123.233,Z 1012.099,A -85,B 0,C 180,E1 22600.643,E2 22600.643} C_VEL
LIN {X 0,Y 138.454,Z 1001.914,A -85,B 0,C 180,E1 22630.457,E2 22630.457} C_VEL
LIN {X 0,Y 182.625,Z 975.285,A -85,B 0,C 180,E1 22653.29,E2 22653.29} C_VEL
LIN {X 0,Y 238.562,Z 934.13,A -85,B 0,C 180,E1 22665.228,E2 22665.228} C_VEL
LIN {X 0,Y 248.595,Z 925.309,A -85,B 0,C 180,E1 22666.925,E2 22666.925} C_VEL
LIN {X 0,Y 194.806,Z 965.016,A -85,B 0,C 180,E1 22677.172,E2 22677.172} C_VEL
LIN {X 0,Y 147.665,Z 991.502,A -85,B 0,C 180,E1 22696.669,E2 22696.669} C_VEL
LIN {X 0,Y 125.846,Z 1002.109,A -85,B 0,C 180,E1 22721.593,E2 22721.593} C_VEL
LIN {X 0,Y 121.723,Z 1002.403,A -85,B 0,C 180,E1 22749.323,E2 22749.323} C_VEL
LIN {X 0,Y 131.818,Z 993.798,A -85,B 0,C 180,E1 22773.301,E2 22773.301} C_VEL
LIN {X 0,Y 153.689,Z 976.993,A -85,B 0,C 180,E1 22792.189,E2 22792.189} C_VEL
LIN {X 0,Y 167.109,Z 962.897,A -85,B 0,C 180,E1 22802.832,E2 22802.832} C_VEL
LIN {X 0,Y 211.476,Z 922.044,A -85,B 0,C 180,E1 22815.126,E2 22815.126} C_VEL
LIN {X 0,Y 235.606,Z 893.659,A -85,B 0,C 180,E1 22819.528,E2 22819.528} C_VEL
LIN {X 0,Y 237.154,Z 877.415,A -85,B 0,C 180,E1 22831.301,E2 22831.301} C_VEL
LIN {X 0,Y 238.199,Z 869.82,A -85,B 0,C 180,E1 22843.32,E2 22843.32} C_VEL
LIN {X 0,Y 239.493,Z 870.793,A -85,B 0,C 180,E1 22852.697,E2 22852.697} C_VEL
LIN {X 0,Y 240.06,Z 882.743,A -85,B 0,C 180,E1 22864.506,E2 22864.506} C_VEL
LIN {X 0,Y 238.376,Z 895.085,A -85,B 0,C 180,E1 22870.956,E2 22870.956} C_VEL
LIN {X 0,Y 193.274,Z 945.898,A -85,B 0,C 180,E1 22879.566,E2 22879.566} C_VEL
LIN {X 0,Y 151.246,Z 981.374,A -85,B 0,C 180,E1 22894.125,E2 22894.125} C_VEL
LIN {X 0,Y 122.216,Z 1003.622,A -85,B 0,C 180,E1 22918.52,E2 22918.52} C_VEL
LIN {X 0,Y 114.968,Z 1011.81,A -85,B 0,C 180,E1 22946.214,E2 22946.214} C_VEL
LIN {X 0,Y 116.665,Z 1010.723,A -85,B 0,C 180,E1 22968.976,E2 22968.976} C_VEL
LIN {X 0,Y 139.511,Z 997.954,A -85,B 0,C 180,E1 22998.545,E2 22998.545} C_VEL
LIN {X 0,Y 190.443,Z 968.609,A -85,B 0,C 180,E1 23018.714,E2 23018.714} C_VEL
LIN {X 0,Y 232.948,Z 938.153,A -85,B 0,C 180,E1 23027.102,E2 23027.102} C_VEL
LIN {X 0,Y 177.077,Z 974.46,A -85,B 0,C 180,E1 23038.935,E2 23038.935} C_VEL
LIN {X 0,Y 132.583,Z 996.522,A -85,B 0,C 180,E1 23061.445,E2 23061.445} C_VEL
LIN {X 0,Y 115.794,Z 1003.349,A -85,B 0,C 180,E1 23086.175,E2 23086.175} C_VEL
LIN {X 0,Y 113.923,Z 1002.536,A -85,B 0,C 180,E1 23110.549,E2 23110.549} C_VEL
LIN {X 0,Y 126.268,Z 992.872,A -85,B 0,C 180,E1 23136.904,E2 23136.904} C_VEL
LIN {X 0,Y 159.951,Z 968.367,A -85,B 0,C 180,E1 23160.05,E2 23160.05} C_VEL
LIN {X 0,Y 167.109,Z 962.897,A -85,B 0,C 180,E1 23162.832,E2 23162.832} C_VEL
LIN {X 0,Y 183.169,Z 946.02,A -85,B 0,C 180,E1 23171.611,E2 23171.611} C_VEL
LIN {X 0,Y 227.975,Z 900.124,A -85,B 0,C 180,E1 23180.572,E2 23180.572} C_VEL
LIN {X 0,Y 230.498,Z 895.199,A -85,B 0,C 180,E1 23182.261,E2 23182.261} C_VEL
LIN {X 0,Y 232.119,Z 881.472,A -85,B 0,C 180,E1 23193.928,E2 23193.928} C_VEL
LIN {X 0,Y 234.064,Z 875.568,A -85,B 0,C 180,E1 23206.863,E2 23206.863} C_VEL
LIN {X 0,Y 234.82,Z 880.038,A -85,B 0,C 180,E1 23216.641,E2 23216.641} C_VEL
LIN {X 0,Y 234.368,Z 894.937,A -85,B 0,C 180,E1 23228.223,E2 23228.223} C_VEL
LIN {X 0,Y 231.725,Z 899.879,A -85,B 0,C 180,E1 23229.656,E2 23229.656} C_VEL
LIN {X 0,Y 187.407,Z 947.638,A -85,B 0,C 180,E1 23237.915,E2 23237.915} C_VEL
LIN {X 0,Y 141.741,Z 984.275,A -85,B 0,C 180,E1 23253.951,E2 23253.951} C_VEL
LIN {X 0,Y 112.123,Z 1005.457,A -85,B 0,C 180,E1 23281.722,E2 23281.722} C_VEL
LIN {X 0,Y 106.958,Z 1011.443,A -85,B 0,C 180,E1 23305.93,E2 23305.93} C_VEL
LIN {X 0,Y 108.95,Z 1010.481,A -85,B 0,C 180,E1 23330.377,E2 23330.377} C_VEL
LIN {X 0,Y 135.427,Z 997.351,A -85,B 0,C 180,E1 23362.023,E2 23362.023} C_VEL
LIN {X 0,Y 190.096,Z 967.685,A -85,B 0,C 180,E1 23381.604,E2 23381.604} C_VEL
LIN {X 0,Y 218.439,Z 948.815,A -85,B 0,C 180,E1 23387.085,E2 23387.085} C_VEL
LIN {X 0,Y 162.693,Z 981.019,A -85,B 0,C 180,E1 23400.002,E2 23400.002} C_VEL
LIN {X 0,Y 122.952,Z 998.462,A -85,B 0,C 180,E1 23422.227,E2 23422.227} C_VEL
LIN {X 0,Y 106.087,Z 1004.108,A -85,B 0,C 180,E1 23451.95,E2 23451.95} C_VEL
LIN {X 0,Y 109.41,Z 1000.207,A -85,B 0,C 180,E1 23482.09,E2 23482.09} C_VEL
LIN {X 0,Y 131.926,Z 984.626,A -85,B 0,C 180,E1 23510.189,E2 23510.189} C_VEL
LIN {X 0,Y 172.933,Z 954.7,A -85,B 0,C 180,E1 23528.703,E2 23528.703} C_VEL
LIN {X 0,Y 183.169,Z 946.02,A -85,B 0,C 180,E1 23531.611,E2 23531.611} C_VEL
LIN {X 0,Y 201.395,Z 926.223,A -85,B 0,C 180,E1 23538.526,E2 23538.526} C_VEL
LIN {X 0,Y 224.917,Z 900.286,A -85,B 0,C 180,E1 23542.925,E2 23542.925} C_VEL
LIN {X 0,Y 227.026,Z 887.28,A -85,B 0,C 180,E1 23554.481,E2 23554.481} C_VEL
LIN {X 0,Y 229.082,Z 881.967,A -85,B 0,C 180,E1 23566.572,E2 23566.572} C_VEL
LIN {X 0,Y 229.663,Z 885.938,A -85,B 0,C 180,E1 23576.187,E2 23576.187} C_VEL
LIN {X 0,Y 228.741,Z 899.656,A -85,B 0,C 180,E1 23587.403,E2 23587.403} C_VEL
LIN {X 0,Y 184.977,Z 946.439,A -85,B 0,C 180,E1 23595.418,E2 23595.418} C_VEL
LIN {X 0,Y 138.31,Z 982.621,A -85,B 0,C 180,E1 23610.434,E2 23610.434} C_VEL
LIN {X 0,Y 107.313,Z 1003.285,A -85,B 0,C 180,E1 23635.549,E2 23635.549} C_VEL
LIN {X 0,Y 98.946,Z 1011.073,A -85,B 0,C 180,E1 23665.6,E2 23665.6} C_VEL
LIN {X 0,Y 101.317,Z 1010.243,A -85,B 0,C 180,E1 23691.989,E2 23691.989} C_VEL
LIN {X 0,Y 130.472,Z 997.458,A -85,B 0,C 180,E1 23724.905,E2 23724.905} C_VEL
LIN {X 0,Y 189.47,Z 967.291,A -85,B 0,C 180,E1 23744.315,E2 23744.315} C_VEL
LIN {X 0,Y 203.552,Z 958.599,A -85,B 0,C 180,E1 23747.097,E2 23747.097} C_VEL
LIN {X 0,Y 146.811,Z 987.415,A -85,B 0,C 180,E1 23761.866,E2 23761.866} C_VEL
LIN {X 0,Y 107.986,Z 1002.052,A -85,B 0,C 180,E1 23789.515,E2 23789.515} C_VEL
LIN {X 0,Y 97.094,Z 1004.269,A -85,B 0,C 180,E1 23819.363,E2 23819.363} C_VEL
LIN {X 0,Y 104.114,Z 998.825,A -85,B 0,C 180,E1 23848.707,E2 23848.707} C_VEL
LIN {X 0,Y 133.166,Z 980.22,A -85,B 0,C 180,E1 23877.121,E2 23877.121} C_VEL
LIN {X 0,Y 177.816,Z 947.692,A -85,B 0,C 180,E1 23893.467,E2 23893.467} C_VEL
LIN {X 0,Y 201.395,Z 926.223,A -85,B 0,C 180,E1 23898.526,E2 23898.526} C_VEL
LIN {X 0,Y 212.54,Z 912.2,A -85,B 0,C 180,E1 23902.949,E2 23902.949} C_VEL
LIN {X 0,Y 219.252,Z 904.695,A -85,B 0,C 180,E1 23903.942,E2 23903.942} C_VEL
LIN {X 0,Y 221.863,Z 892.483,A -85,B 0,C 180,E1 23915.88,E2 23915.88} C_VEL
LIN {X 0,Y 224.317,Z 888.299,A -85,B 0,C 180,E1 23928.812,E2 23928.812} C_VEL
LIN {X 0,Y 224.146,Z 896.082,A -85,B 0,C 180,E1 23940.286,E2 23940.286} C_VEL
LIN {X 0,Y 222.38,Z 904.977,A -85,B 0,C 180,E1 23946.385,E2 23946.385} C_VEL
LIN {X 0,Y 174.661,Z 952.177,A -85,B 0,C 180,E1 23954.645,E2 23954.645} C_VEL
LIN {X 0,Y 127.884,Z 985.861,A -85,B 0,C 180,E1 23970.442,E2 23970.442} C_VEL
LIN {X 0,Y 96.569,Z 1005.34,A -85,B 0,C 180,E1 23999.65,E2 23999.65} C_VEL
LIN {X 0,Y 90.929,Z 1010.697,A -85,B 0,C 180,E1 24025.211,E2 24025.211} C_VEL
LIN {X 0,Y 93.762,Z 1010.01,A -85,B 0,C 180,E1 24053.866,E2 24053.866} C_VEL
LIN {X 0,Y 125.85,Z 997.557,A -85,B 0,C 180,E1 24087.998,E2 24087.998} C_VEL
LIN {X 0,Y 188.237,Z 967.514,A -85,B 0,C 180,E1 24107.152,E2 24107.152} C_VEL
LIN {X 0,Y 129.439,Z 993.43,A -85,B 0,C 180,E1 24124.764,E2 24124.764} C_VEL
LIN {X 0,Y 96.909,Z 1003.612,A -85,B 0,C 180,E1 24153.296,E2 24153.296} C_VEL
LIN {X 0,Y 89.409,Z 1003.653,A -85,B 0,C 180,E1 24189.126,E2 24189.126} C_VEL
LIN {X 0,Y 101.846,Z 995.911,A -85,B 0,C 180,E1 24218.677,E2 24218.677} C_VEL
LIN {X 0,Y 139.685,Z 973.064,A -85,B 0,C 180,E1 24245.166,E2 24245.166} C_VEL
LIN {X 0,Y 187.159,Z 936.96,A -85,B 0,C 180,E1 24258.596,E2 24258.596} C_VEL
LIN {X 0,Y 212.54,Z 912.2,A -85,B 0,C 180,E1 24262.949,E2 24262.949} C_VEL
LIN {X 0,Y 215.213,Z 906.371,A -85,B 0,C 180,E1 24266.352,E2 24266.352} C_VEL
LIN {X 0,Y 214.975,Z 904.314,A -85,B 0,C 180,E1 24268.993,E2 24268.993} C_VEL
LIN {X 0,Y 217.499,Z 895.616,A -85,B 0,C 180,E1 24281.679,E2 24281.679} C_VEL
LIN {X 0,Y 219.289,Z 895.332,A -85,B 0,C 180,E1 24291.855,E2 24291.855} C_VEL
LIN {X 0,Y 217.988,Z 906.002,A -85,B 0,C 180,E1 24303.497,E2 24303.497} C_VEL
LIN {X 0,Y 214.303,Z 911.387,A -85,B 0,C 180,E1 24305.132,E2 24305.132} C_VEL
LIN {X 0,Y 165.745,Z 956.448,A -85,B 0,C 180,E1 24313.426,E2 24313.426} C_VEL
LIN {X 0,Y 118.243,Z 988.413,A -85,B 0,C 180,E1 24329.962,E2 24329.962} C_VEL
LIN {X 0,Y 86.391,Z 1006.803,A -85,B 0,C 180,E1 24363.947,E2 24363.947} C_VEL
LIN {X 0,Y 83.036,Z 1010.883,A -85,B 0,C 180,E1 24395.241,E2 24395.241} C_VEL
LIN {X 0,Y 97.746,Z 1006.031,A -85,B 0,C 180,E1 24434.317,E2 24434.317} C_VEL
LIN {X 0,Y 151.586,Z 985.427,A -85,B 0,C 180,E1 24462.002,E2 24462.002} C_VEL
LIN {X 0,Y 172.276,Z 975.62,A -85,B 0,C 180,E1 24467.318,E2 24467.318} C_VEL
LIN {X 0,Y 114.681,Z 997.544,A -85,B 0,C 180,E1 24487.042,E2 24487.042} C_VEL
LIN {X 0,Y 85.855,Z 1004.746,A -85,B 0,C 180,E1 24518.291,E2 24518.291} C_VEL
LIN {X 0,Y 82.19,Z 1003.359,A -85,B 0,C 180,E1 24553.923,E2 24553.923} C_VEL
LIN {X 0,Y 100.915,Z 992.979,A -85,B 0,C 180,E1 24587.505,E2 24587.505} C_VEL
LIN {X 0,Y 144.429,Z 967.474,A -85,B 0,C 180,E1 24611.052,E2 24611.052} C_VEL
LIN {X 0,Y 193.608,Z 928.783,A -85,B 0,C 180,E1 24622.529,E2 24622.529} C_VEL
LIN {X 0,Y 213.958,Z 908.123,A -85,B 0,C 180,E1 24625.746,E2 24625.746} C_VEL
LIN {X 0,Y 214.975,Z 904.314,A -85,B 0,C 180,E1 24628.993,E2 24628.993} C_VEL
LIN {X 0,Y 211.347,Z 903.003,A -85,B 0,C 180,E1 24638.561,E2 24638.561} C_VEL
LIN {X 0,Y 213.96,Z 900.417,A -85,B 0,C 180,E1 24649.762,E2 24649.762} C_VEL
LIN {X 0,Y 212.443,Z 909.98,A -85,B 0,C 180,E1 24662.018,E2 24662.018} C_VEL
LIN {X 0,Y 210.249,Z 913.356,A -85,B 0,C 180,E1 24663.28,E2 24663.28} C_VEL
LIN {X 0,Y 160.547,Z 957.796,A -85,B 0,C 180,E1 24671.267,E2 24671.267} C_VEL
LIN {X 0,Y 111.478,Z 989.162,A -85,B 0,C 180,E1 24687.761,E2 24687.761} C_VEL
LIN {X 0,Y 79.1,Z 1006.305,A -85,B 0,C 180,E1 24721.335,E2 24721.335} C_VEL
LIN {X 0,Y 75,Z 1010.551,A -85,B 0,C 180,E1 24755.804,E2 24755.804} C_VEL
LIN {X 0,Y 91.999,Z 1005.947,A -85,B 0,C 180,E1 24797.925,E2 24797.925} C_VEL
LIN {X 0,Y 149.238,Z 985.879,A -85,B 0,C 180,E1 24825.023,E2 24825.023} C_VEL
LIN {X 0,Y 157.933,Z 982.075,A -85,B 0,C 180,E1 24827.169,E2 24827.169} C_VEL
LIN {X 0,Y 100.157,Z 1000.859,A -85,B 0,C 180,E1 24849.985,E2 24849.985} C_VEL
LIN {X 0,Y 75.054,Z 1005.407,A -85,B 0,C 180,E1 24885.139,E2 24885.139} C_VEL
LIN {X 0,Y 77.223,Z 1002.018,A -85,B 0,C 180,E1 24924.363,E2 24924.363} C_VEL
LIN {X 0,Y 106.99,Z 986.923,A -85,B 0,C 180,E1 24959.768,E2 24959.768} C_VEL
LIN {X 0,Y 157.194,Z 956.491,A -85,B 0,C 180,E1 24978.437,E2 24978.437} C_VEL
LIN {X 0,Y 207.815,Z 912.815,A -85,B 0,C 180,E1 24987.121,E2 24987.121} C_VEL
LIN {X 0,Y 211.025,Z 903.924,A -85,B 0,C 180,E1 24996.679,E2 24996.679} C_VEL
LIN {X 0,Y 211.347,Z 903.003,A -85,B 0,C 180,E1 24998.561,E2 24998.561} C_VEL
LIN {X 0,Y 207.966,Z 906.294,A -85,B 0,C 180,E1 25008.258,E2 25008.258} C_VEL
LIN {X 0,Y 207.249,Z 912.514,A -85,B 0,C 180,E1 25019.028,E2 25019.028} C_VEL
LIN {X 0,Y 204.95,Z 916.765,A -85,B 0,C 180,E1 25021.519,E2 25021.519} C_VEL
LIN {X 0,Y 151.631,Z 961.955,A -85,B 0,C 180,E1 25029.797,E2 25029.797} C_VEL
LIN {X 0,Y 98.434,Z 993.035,A -85,B 0,C 180,E1 25048.843,E2 25048.843} C_VEL
LIN {X 0,Y 69.792,Z 1007.05,A -85,B 0,C 180,E1 25084.219,E2 25084.219} C_VEL
LIN {X 0,Y 66.993,Z 1010.219,A -85,B 0,C 180,E1 25116.501,E2 25116.501} C_VEL
LIN {X 0,Y 87.44,Z 1005.663,A -85,B 0,C 180,E1 25162.695,E2 25162.695} C_VEL
LIN {X 0,Y 142.299,Z 988.203,A -85,B 0,C 180,E1 25186.994,E2 25186.994} C_VEL
LIN {X 0,Y 85.884,Z 1003.389,A -85,B 0,C 180,E1 25213.634,E2 25213.634} C_VEL
LIN {X 0,Y 65.086,Z 1005.485,A -85,B 0,C 180,E1 25254.823,E2 25254.823} C_VEL
LIN {X 0,Y 74.002,Z 1000.143,A -85,B 0,C 180,E1 25295.888,E2 25295.888} C_VEL
LIN {X 0,Y 111.07,Z 982.564,A -85,B 0,C 180,E1 25327.943,E2 25327.943} C_VEL
LIN {X 0,Y 163.566,Z 949.993,A -85,B 0,C 180,E1 25343.074,E2 25343.074} C_VEL
LIN {X 0,Y 203.161,Z 915.584,A -85,B 0,C 180,E1 25349.211,E2 25349.211} C_VEL
LIN {X 0,Y 206.187,Z 907.815,A -85,B 0,C 180,E1 25360.634,E2 25360.634} C_VEL
LIN {X 0,Y 207.966,Z 906.294,A -85,B 0,C 180,E1 25368.258,E2 25368.258} C_VEL
LIN {X 0,Y 205.384,Z 910.567,A -85,B 0,C 180,E1 25372.922,E2 25372.922} C_VEL
LIN {X 0,Y 201.623,Z 916.943,A -85,B 0,C 180,E1 25377.683,E2 25377.683} C_VEL
LIN {X 0,Y 199.376,Z 920.372,A -85,B 0,C 180,E1 25379.708,E2 25379.708} C_VEL
LIN {X 0,Y 147,Z 962.982,A -85,B 0,C 180,E1 25387.271,E2 25387.271} C_VEL
LIN {X 0,Y 92.543,Z 993.245,A -85,B 0,C 180,E1 25405.583,E2 25405.583} C_VEL
LIN {X 0,Y 60.608,Z 1007.609,A -85,B 0,C 180,E1 25447.936,E2 25447.936} C_VEL
LIN {X 0,Y 58.966,Z 1009.883,A -85,B 0,C 180,E1 25477.39,E2 25477.39} C_VEL
LIN {X 0,Y 81.808,Z 1005.826,A -85,B 0,C 180,E1 25526.588,E2 25526.588} C_VEL
LIN {X 0,Y 126.032,Z 993.639,A -85,B 0,C 180,E1 25546.847,E2 25546.847} C_VEL
LIN {X 0,Y 84.016,Z 1003.326,A -85,B 0,C 180,E1 25566.568,E2 25566.568} C_VEL
LIN {X 0,Y 57.713,Z 1005.917,A -85,B 0,C 180,E1 25608.903,E2 25608.903} C_VEL
LIN {X 0,Y 65.648,Z 1000.869,A -85,B 0,C 180,E1 25656.64,E2 25656.64} C_VEL
LIN {X 0,Y 104.791,Z 983.857,A -85,B 0,C 180,E1 25690.672,E2 25690.672} C_VEL
LIN {X 0,Y 159.511,Z 951.366,A -85,B 0,C 180,E1 25705.5,E2 25705.5} C_VEL
LIN {X 0,Y 197.671,Z 919.582,A -85,B 0,C 180,E1 25710.846,E2 25710.846} C_VEL
LIN {X 0,Y 200.61,Z 913.402,A -85,B 0,C 180,E1 25721.019,E2 25721.019} C_VEL
LIN {X 0,Y 202.637,Z 911.959,A -85,B 0,C 180,E1 25729.183,E2 25729.183} C_VEL
LIN {X 0,Y 201.623,Z 916.943,A -85,B 0,C 180,E1 25737.683,E2 25737.683} C_VEL
LIN {X 0,Y 194.94,Z 923.818,A -85,B 0,C 180,E1 25738.872,E2 25738.872} C_VEL
LIN {X 0,Y 184.105,Z 932.9,A -85,B 0,C 180,E1 25738.815,E2 25738.815} C_VEL
LIN {X 0,Y 128.184,Z 972.747,A -85,B 0,C 180,E1 25747.454,E2 25747.454} C_VEL
LIN {X 0,Y 77.304,Z 997.402,A -85,B 0,C 180,E1 25767.937,E2 25767.937} C_VEL
LIN {X 0,Y 53.174,Z 1007.146,A -85,B 0,C 180,E1 25804.649,E2 25804.649} C_VEL
LIN {X 0,Y 50.964,Z 1009.548,A -85,B 0,C 180,E1 25838.559,E2 25838.559} C_VEL
LIN {X 0,Y 77.539,Z 1005.762,A -85,B 0,C 180,E1 25891.727,E2 25891.727} C_VEL
LIN {X 0,Y 111.202,Z 997.747,A -85,B 0,C 180,E1 25907.452,E2 25907.452} C_VEL
LIN {X 0,Y 58.17,Z 1006.297,A -85,B 0,C 180,E1 25944.069,E2 25944.069} C_VEL
LIN {X 0,Y 51.044,Z 1003.936,A -85,B 0,C 180,E1 26001.455,E2 26001.455} C_VEL
LIN {X 0,Y 78.463,Z 993.713,A -85,B 0,C 180,E1 26042.464,E2 26042.464} C_VEL
LIN {X 0,Y 132.141,Z 967.823,A -85,B 0,C 180,E1 26063.509,E2 26063.509} C_VEL
LIN {X 0,Y 186.5,Z 928.621,A -85,B 0,C 180,E1 26072.057,E2 26072.057} C_VEL
LIN {X 0,Y 192.314,Z 923.405,A -85,B 0,C 180,E1 26072.828,E2 26072.828} C_VEL
LIN {X 0,Y 195.872,Z 917.783,A -85,B 0,C 180,E1 26085.581,E2 26085.581} C_VEL
LIN {X 0,Y 196.076,Z 920.728,A -85,B 0,C 180,E1 26095.532,E2 26095.532} C_VEL
LIN {X 0,Y 193.329,Z 924.615,A -85,B 0,C 180,E1 26097.864,E2 26097.864} C_VEL
LIN {X 0,Y 184.105,Z 932.9,A -85,B 0,C 180,E1 26098.815,E2 26098.815} C_VEL
LIN {X 0,Y 155.48,Z 953.869,A -85,B 0,C 180,E1 26099.317,E2 26099.317} C_VEL
LIN {X 0,Y 97.059,Z 987.059,A -85,B 0,C 180,E1 26111.487,E2 26111.487} C_VEL
LIN {X 0,Y 49.976,Z 1005.07,A -85,B 0,C 180,E1 26149.185,E2 26149.185} C_VEL
LIN {X 0,Y 42.972,Z 1009.21,A -85,B 0,C 180,E1 26200.166,E2 26200.166} C_VEL
LIN {X 0,Y 73.952,Z 1005.649,A -85,B 0,C 180,E1 26257.43,E2 26257.43} C_VEL
LIN {X 0,Y 95.441,Z 1001.359,A -85,B 0,C 180,E1 26267.448,E2 26267.448} C_VEL
LIN {X 0,Y 46.268,Z 1006.741,A -85,B 0,C 180,E1 26309.608,E2 26309.608} C_VEL
LIN {X 0,Y 48.77,Z 1002.307,A -85,B 0,C 180,E1 26378.955,E2 26378.955} C_VEL
LIN {X 0,Y 93.101,Z 986.164,A -85,B 0,C 180,E1 26417.186,E2 26417.186} C_VEL
LIN {X 0,Y 148.664,Z 956.437,A -85,B 0,C 180,E1 26430.194,E2 26430.194} C_VEL
LIN {X 0,Y 186.753,Z 927.333,A -85,B 0,C 180,E1 26434.802,E2 26434.802} C_VEL
LIN {X 0,Y 190.712,Z 923.02,A -85,B 0,C 180,E1 26448.498,E2 26448.498} C_VEL
LIN {X 0,Y 188.976,Z 927.159,A -85,B 0,C 180,E1 26455.778,E2 26455.778} C_VEL
LIN {X 0,Y 155.48,Z 953.869,A -85,B 0,C 180,E1 26459.317,E2 26459.317} C_VEL
LIN {X 0,Y 124.812,Z 971.665,A -85,B 0,C 180,E1 26460.249,E2 26460.249} C_VEL
LIN {X 0,Y 66.169,Z 997.525,A -85,B 0,C 180,E1 26478.69,E2 26478.69} C_VEL
LIN {X 0,Y 34.977,Z 1007.923,A -85,B 0,C 180,E1 26537.465,E2 26537.465} C_VEL
LIN {X 0,Y 38.905,Z 1008.971,A -85,B 0,C 180,E1 26585.805,E2 26585.805} C_VEL
LIN {X 0,Y 78.118,Z 1004.396,A -85,B 0,C 180,E1 26628.06,E2 26628.06} C_VEL
LIN {X 0,Y 40.686,Z 1007.068,A -85,B 0,C 180,E1 26661.184,E2 26661.184} C_VEL
LIN {X 0,Y 40.251,Z 1003.022,A -85,B 0,C 180,E1 26740.871,E2 26740.871} C_VEL
LIN {X 0,Y 83.158,Z 989.142,A -85,B 0,C 180,E1 26779.327,E2 26779.327} C_VEL
LIN {X 0,Y 142.998,Z 959.281,A -85,B 0,C 180,E1 26792.727,E2 26792.727} C_VEL
LIN {X 0,Y 180.522,Z 932.084,A -85,B 0,C 180,E1 26796.66,E2 26796.66} C_VEL
LIN {X 0,Y 184.475,Z 928.328,A -85,B 0,C 180,E1 26808.103,E2 26808.103} C_VEL
LIN {X 0,Y 183.195,Z 931.085,A -85,B 0,C 180,E1 26813.718,E2 26813.718} C_VEL
LIN {X 0,Y 127.013,Z 970.448,A -85,B 0,C 180,E1 26819.88,E2 26819.88} C_VEL
LIN {X 0,Y 124.812,Z 971.665,A -85,B 0,C 180,E1 26820.249,E2 26820.249} C_VEL
LIN {X 0,Y 92.591,Z 986.177,A -85,B 0,C 180,E1 26822.051,E2 26822.051} C_VEL
LIN {X 0,Y 42.908,Z 1002.902,A -85,B 0,C 180,E1 26847.837,E2 26847.837} C_VEL
LIN {X 0,Y 27.135,Z 1007.434,A -85,B 0,C 180,E1 26893.754,E2 26893.754} C_VEL
LIN {X 0,Y 34.538,Z 1008.628,A -85,B 0,C 180,E1 26959.014,E2 26959.014} C_VEL
LIN {X 0,Y 62.78,Z 1006.324,A -85,B 0,C 180,E1 26987.619,E2 26987.619} C_VEL
LIN {X 0,Y 27.239,Z 1006.978,A -85,B 0,C 180,E1 27033.323,E2 27033.323} C_VEL
LIN {X 0,Y 42.927,Z 1000.961,A -85,B 0,C 180,E1 27122.03,E2 27122.03} C_VEL
LIN {X 0,Y 100.884,Z 981.005,A -85,B 0,C 180,E1 27149.883,E2 27149.883} C_VEL
LIN {X 0,Y 159.517,Z 947.634,A -85,B 0,C 180,E1 27157.668,E2 27157.668} C_VEL
LIN {X 0,Y 175.453,Z 935.615,A -85,B 0,C 180,E1 27159.075,E2 27159.075} C_VEL
LIN {X 0,Y 178.218,Z 934.397,A -85,B 0,C 180,E1 27171.278,E2 27171.278} C_VEL
LIN {X 0,Y 119.075,Z 973.672,A -85,B 0,C 180,E1 27177.156,E2 27177.156} C_VEL
LIN {X 0,Y 92.591,Z 986.177,A -85,B 0,C 180,E1 27182.051,E2 27182.051} C_VEL
LIN {X 0,Y 59.04,Z 997.087,A -85,B 0,C 180,E1 27185.56,E2 27185.56} C_VEL
LIN {X 0,Y 19.504,Z 1006.937,A -85,B 0,C 180,E1 27247.094,E2 27247.094} C_VEL
LIN {X 0,Y 27.375,Z 1008.275,A -85,B 0,C 180,E1 27326.246,E2 27326.246} C_VEL
LIN {X 0,Y 44.786,Z 1007.653,A -85,B 0,C 180,E1 27347.637,E2 27347.637} C_VEL
LIN {X 0,Y 16.266,Z 1006.27,A -85,B 0,C 180,E1 27422.206,E2 27422.206} C_VEL
LIN {X 0,Y 49.828,Z 998.376,A -85,B 0,C 180,E1 27499.594,E2 27499.594} C_VEL
LIN {X 0,Y 114.509,Z 974.211,A -85,B 0,C 180,E1 27516.33,E2 27516.33} C_VEL
LIN {X 0,Y 169.854,Z 939.735,A -85,B 0,C 180,E1 27521.747,E2 27521.747} C_VEL
LIN {X 0,Y 171.939,Z 938.648,A -85,B 0,C 180,E1 27528.798,E2 27528.798} C_VEL
LIN {X 0,Y 114.514,Z 975.176,A -85,B 0,C 180,E1 27533.699,E2 27533.699} C_VEL
LIN {X 0,Y 59.04,Z 997.087,A -85,B 0,C 180,E1 27545.56,E2 27545.56} C_VEL
LIN {X 0,Y 24.898,Z 1004.224,A -85,B 0,C 180,E1 27556.203,E2 27556.203} C_VEL
LIN {X 0,Y 12.44,Z 1007.575,A -85,B 0,C 180,E1 27667.569,E2 27667.569} C_VEL
LIN {X 0,Y 24.545,Z 1007.861,A -85,B 0,C 180,E1 27707.867,E2 27707.867} C_VEL
LIN {X 0,Y 29.982,Z 1002.403,A -85,B 0,C 180,E1 27859.408,E2 27859.408} C_VEL
LIN {X 0,Y 90.01,Z 984.869,A -85,B 0,C 180,E1 27878.025,E2 27878.025} C_VEL
LIN {X 0,Y 152.552,Z 952.115,A -85,B 0,C 180,E1 27883.133,E2 27883.133} C_VEL
LIN {X 0,Y 163.035,Z 944.794,A -85,B 0,C 180,E1 27883.652,E2 27883.652} C_VEL
LIN {X 0,Y 163.635,Z 944.614,A -85,B 0,C 180,E1 27886.86,E2 27886.86} C_VEL
LIN {X 0,Y 103.86,Z 979.575,A -85,B 0,C 180,E1 27890.515,E2 27890.515} C_VEL
LIN {X 0,Y 45.004,Z 1000.017,A -85,B 0,C 180,E1 27901.896,E2 27901.896} C_VEL
LIN {X 0,Y 24.898,Z 1004.224,A -85,B 0,C 180,E1 27916.203,E2 27916.203} C_VEL
LIN {X 0,Y 1.179,Z 1006.539,A -85,B 0,C 180,E1 27946.565,E2 27946.565} C_VEL
LIN {X 0,Y 36.489,Z 1000.879,A -85,B 0,C 180,E1 27876.567,E2 27876.567} C_VEL
LIN {X 0,Y 102.673,Z 979.604,A -85,B 0,C 180,E1 27883.9,E2 27883.9} C_VEL
LIN {X 0,Y 117.575,Z 972.603,A -85,B 0,C 180,E1 27885.485,E2 27885.485} C_VEL
LIN {X 0,Y 53.92,Z 997.042,A -85,B 0,C 180,E1 27890.111,E2 27890.111} C_VEL
LIN {X 0,Y 5.028,Z 1006.227,A -85,B 0,C 180,E1 27922.087,E2 27922.087} C_VEL
LIN {X 0,Y 1.179,Z 1006.539,A -85,B 0,C 180,E1 27946.565,E2 27946.565} C_VEL
LIN {X 0,Y 1.041,Z 1008.533,A -85,B 0,C 180,E1 28058.731,E2 28058.731} C_VEL
LIN {X 0,Y 1.041,Z 1028,A -85,B 0,C 180,E1 28058.731,E2 28058.731} C_VEL
LIN {X 0,Y 1.041,Z 1028,A -85,B 0,C 180,E1 28058.731,E2 28058.731}

QRS_NEXT_CUT()
PTP {E1 27896.858,E2 27896.858}
PTP {X 0,Y 607.913,A -85,B 0,C 180,E1 27896.858,E2 27896.858,E3 0,E4 0,E5 0,E6 0}
QRS_SPEED_INIT()
LIN {X 0,Y 607.913,Z 1028,A -85,B 0,C 180,E1 27896.858,E2 27896.858,E3 0,E4 0,E5 0,E6 0} C_VEL
LIN {X 0,Y 607.913,Z 365.4,A -85,B 0,C 180,E1 27896.858,E2 27896.858} C_VEL
LIN {X 0,Y 607.913,Z 357.323,A -85,B 0,C 180,E1 27896.858,E2 27896.858} C_VEL
LIN {X 0,Y 607.886,Z 355.323,A -85,B 0,C 180,E1 27896.669,E2 27896.669} C_VEL
LIN {X 0,Y 607.848,Z 355.325,A -85,B 0,C 180,E1 27893.767,E2 27893.767} C_VEL
LIN {X 0,Y 607.909,Z 355.322,A -85,B 0,C 180,E1 27890.628,E2 27890.628} C_VEL
LIN {X 0,Y 607.851,Z 355.325,A -85,B 0,C 180,E1 27887.652,E2 27887.652} C_VEL
LIN {X 0,Y 607.919,Z 355.321,A -85,B 0,C 180,E1 27884.519,E2 27884.519} C_VEL
LIN {X 0,Y 607.855,Z 355.324,A -85,B 0,C 180,E1 27881.49,E2 27881.49} C_VEL
LIN {X 0,Y 607.914,Z 355.322,A -85,B 0,C 180,E1 27878.381,E2 27878.381} C_VEL
LIN {X 0,Y 607.858,Z 355.324,A -85,B 0,C 180,E1 27875.304,E2 27875.304} C_VEL
LIN {X 0,Y 607.917,Z 355.32,A -85,B 0,C 180,E1 27872.153,E2 27872.153} C_VEL
LIN {X 0,Y 607.863,Z 355.324,A -85,B 0,C 180,E1 27869.122,E2 27869.122} C_VEL
LIN {X 0,Y 607.916,Z 355.32,A -85,B 0,C 180,E1 27865.982,E2 27865.982} C_VEL
LIN {X 0,Y 607.868,Z 355.324,A -85,B 0,C 180,E1 27862.909,E2 27862.909} C_VEL
LIN {X 0,Y 607.917,Z 355.319,A -85,B 0,C 180,E1 27859.73,E2 27859.73} C_VEL
LIN {X 0,Y 607.878,Z 355.324,A -85,B 0,C 180,E1 27856.564,E2 27856.564} C_VEL
LIN {X 0,Y 607.9,Z 355.318,A -85,B 0,C 180,E1 27853.298,E2 27853.298} C_VEL
LIN {X 0,Y 607.903,Z 355.326,A -85,B 0,C 180,E1 27850.109,E2 27850.109} C_VEL
LIN {X 0,Y 607.886,Z 355.32,A -85,B 0,C 180,E1 27846.89,E2 27846.89} C_VEL
LIN {X 0,Y 607.911,Z 355.327,A -85,B 0,C 180,E1 27843.769,E2 27843.769} C_VEL
LIN {X 0,Y 607.882,Z 355.32,A -85,B 0,C 180,E1 27840.543,E2 27840.543} C_VEL
LIN {X 0,Y 607.908,Z 355.324,A -85,B 0,C 180,E1 27837.417,E2 27837.417} C_VEL
LIN {X 0,Y 607.883,Z 355.32,A -85,B 0,C 180,E1 27834.276,E2 27834.276} C_VEL
LIN {X 0,Y 607.904,Z 355.322,A -85,B 0,C 180,E1 27831.109,E2 27831.109} C_VEL
LIN {X 0,Y 607.885,Z 355.322,A -85,B 0,C 180,E1 27828.009,E2 27828.009} C_VEL
LIN {X 0,Y 607.903,Z 355.323,A -85,B 0,C 180,E1 27824.961,E2 27824.961} C_VEL
LIN {X 0,Y 607.888,Z 355.317,A -85,B 0,C 180,E1 27821.856,E2 27821.856} C_VEL
LIN {X 0,Y 607.888,Z 355.422,A -85,B 0,C 180,E1 27819.751,E2 27819.751} C_VEL
LIN {X 0,Y 607.906,Z 361.67,A -85,B 0,C 180,E1 27819.316,E2 27819.316} C_VEL
LIN {X 0,Y 607.92,Z 559.871,A -85,B 0,C 180,E1 27816.478,E2 27816.478} C_VEL
LIN {X 0,Y 607.914,Z 708.935,A -85,B 0,C 180,E1 27814.383,E2 27814.383} C_VEL
LIN {X 0,Y 607.915,Z 732.02,A -85,B 0,C 180,E1 27813.887,E2 27813.887} C_VEL
LIN {X 0,Y 607.915,Z 751.443,A -85,B 0,C 180,E1 27813.321,E2 27813.321} C_VEL
LIN {X 0,Y 607.912,Z 772.885,A -85,B 0,C 180,E1 27812.542,E2 27812.542} C_VEL
LIN {X 0,Y 607.918,Z 792.829,A -85,B 0,C 180,E1 27811.646,E2 27811.646} C_VEL
LIN {X 0,Y 607.916,Z 813.472,A -85,B 0,C 180,E1 27810.563,E2 27810.563} C_VEL
LIN {X 0,Y 607.914,Z 833.866,A -85,B 0,C 180,E1 27809.29,E2 27809.29} C_VEL
LIN {X 0,Y 607.916,Z 854.171,A -85,B 0,C 180,E1 27807.829,E2 27807.829} C_VEL
LIN {X 0,Y 607.905,Z 872.447,A -85,B 0,C 180,E1 27806.319,E2 27806.319} C_VEL
LIN {X 0,Y 607.903,Z 889.422,A -85,B 0,C 180,E1 27804.713,E2 27804.713} C_VEL
LIN {X 0,Y 607.904,Z 905.394,A -85,B 0,C 180,E1 27803.006,E2 27803.006} C_VEL
LIN {X 0,Y 607.906,Z 920.138,A -85,B 0,C 180,E1 27801.199,E2 27801.199} C_VEL
LIN {X 0,Y 607.908,Z 934.423,A -85,B 0,C 180,E1 27799.19,E2 27799.19} C_VEL
LIN {X 0,Y 607.912,Z 946.401,A -85,B 0,C 180,E1 27797.249,E2 27797.249} C_VEL
LIN {X 0,Y 607.906,Z 956.946,A -85,B 0,C 180,E1 27795.228,E2 27795.228} C_VEL
LIN {X 0,Y 607.896,Z 966.088,A -85,B 0,C 180,E1 27793.171,E2 27793.171} C_VEL
LIN {X 0,Y 607.917,Z 973.48,A -85,B 0,C 180,E1 27791.092,E2 27791.092} C_VEL
LIN {X 0,Y 607.902,Z 979.5,A -85,B 0,C 180,E1 27788.986,E2 27788.986} C_VEL
LIN {X 0,Y 607.894,Z 983.826,A -85,B 0,C 180,E1 27786.845,E2 27786.845} C_VEL
LIN {X 0,Y 607.913,Z 986.725,A -85,B 0,C 180,E1 27784.681,E2 27784.681} C_VEL
LIN {X 0,Y 607.89,Z 987.859,A -85,B 0,C 180,E1 27782.576,E2 27782.576} C_VEL
LIN {X 0,Y 607.896,Z 987.581,A -85,B 0,C 180,E1 27780.431,E2 27780.431} C_VEL
LIN {X 0,Y 607.902,Z 985.798,A -85,B 0,C 180,E1 27778.43,E2 27778.43} C_VEL
LIN {X 0,Y 607.884,Z 982.583,A -85,B 0,C 180,E1 27776.334,E2 27776.334} C_VEL
LIN {X 0,Y 607.915,Z 977.759,A -85,B 0,C 180,E1 27774.274,E2 27774.274} C_VEL
LIN {X 0,Y 607.893,Z 971.306,A -85,B 0,C 180,E1 27772.14,E2 27772.14} C_VEL
LIN {X 0,Y 607.893,Z 963.356,A -85,B 0,C 180,E1 27770.097,E2 27770.097} C_VEL
LIN {X 0,Y 607.914,Z 953.762,A -85,B 0,C 180,E1 27768.024,E2 27768.024} C_VEL
LIN {X 0,Y 607.904,Z 942.737,A -85,B 0,C 180,E1 27766.043,E2 27766.043} C_VEL
LIN {X 0,Y 607.899,Z 929.896,A -85,B 0,C 180,E1 27764.045,E2 27764.045} C_VEL
LIN {X 0,Y 607.91,Z 916.587,A -85,B 0,C 180,E1 27762.255,E2 27762.255} C_VEL
LIN {X 0,Y 607.918,Z 900.215,A -85,B 0,C 180,E1 27760.331,E2 27760.331} C_VEL
LIN {X 0,Y 607.912,Z 883.65,A -85,B 0,C 180,E1 27758.623,E2 27758.623} C_VEL
LIN {X 0,Y 607.912,Z 866.576,A -85,B 0,C 180,E1 27757.087,E2 27757.087} C_VEL
LIN {X 0,Y 607.91,Z 846.347,A -85,B 0,C 180,E1 27755.493,E2 27755.493} C_VEL
LIN {X 0,Y 607.918,Z 827.168,A -85,B 0,C 180,E1 27754.176,E2 27754.176} C_VEL
LIN {X 0,Y 607.916,Z 806.813,A -85,B 0,C 180,E1 27752.983,E2 27752.983} C_VEL
LIN {X 0,Y 607.916,Z 785.924,A -85,B 0,C 180,E1 27751.93,E2 27751.93} C_VEL
LIN {X 0,Y 607.913,Z 764.87,A -85,B 0,C 180,E1 27751.061,E2 27751.061} C_VEL
LIN {X 0,Y 607.916,Z 744.97,A -85,B 0,C 180,E1 27750.382,E2 27750.382} C_VEL
LIN {X 0,Y 607.914,Z 723.136,A -85,B 0,C 180,E1 27749.81,E2 27749.81} C_VEL
LIN {X 0,Y 607.912,Z 703.889,A -85,B 0,C 180,E1 27749.444,E2 27749.444} C_VEL
LIN {X 0,Y 607.919,Z 478.822,A -85,B 0,C 180,E1 27746.286,E2 27746.286} C_VEL
LIN {X 0,Y 607.917,Z 361.185,A -85,B 0,C 180,E1 27744.574,E2 27744.574} C_VEL
LIN {X 0,Y 607.912,Z 355.574,A -85,B 0,C 180,E1 27744.137,E2 27744.137} C_VEL
LIN {X 0,Y 607.876,Z 355.323,A -85,B 0,C 180,E1 27741.15,E2 27741.15} C_VEL
LIN {X 0,Y 607.909,Z 355.323,A -85,B 0,C 180,E1 27738.012,E2 27738.012} C_VEL
LIN {X 0,Y 607.883,Z 355.322,A -85,B 0,C 180,E1 27734.868,E2 27734.868} C_VEL
LIN {X 0,Y 607.903,Z 355.321,A -85,B 0,C 180,E1 27731.768,E2 27731.768} C_VEL
LIN {X 0,Y 607.891,Z 355.322,A -85,B 0,C 180,E1 27728.685,E2 27728.685} C_VEL
LIN {X 0,Y 607.898,Z 355.32,A -85,B 0,C 180,E1 27725.569,E2 27725.569} C_VEL
LIN {X 0,Y 607.903,Z 355.325,A -85,B 0,C 180,E1 27722.357,E2 27722.357} C_VEL
LIN {X 0,Y 607.903,Z 355.318,A -85,B 0,C 180,E1 27719.152,E2 27719.152} C_VEL
LIN {X 0,Y 607.901,Z 355.326,A -85,B 0,C 180,E1 27715.85,E2 27715.85} C_VEL
LIN {X 0,Y 607.912,Z 355.318,A -85,B 0,C 180,E1 27712.63,E2 27712.63} C_VEL
LIN {X 0,Y 607.879,Z 355.324,A -85,B 0,C 180,E1 27709.481,E2 27709.481} C_VEL
LIN {X 0,Y 607.913,Z 355.32,A -85,B 0,C 180,E1 27706.397,E2 27706.397} C_VEL
LIN {X 0,Y 607.869,Z 355.324,A -85,B 0,C 180,E1 27703.271,E2 27703.271} C_VEL
LIN {X 0,Y 607.915,Z 355.322,A -85,B 0,C 180,E1 27700.186,E2 27700.186} C_VEL
LIN {X 0,Y 607.858,Z 355.324,A -85,B 0,C 180,E1 27697.056,E2 27697.056} C_VEL
LIN {X 0,Y 607.914,Z 355.323,A -85,B 0,C 180,E1 27694.056,E2 27694.056} C_VEL
LIN {X 0,Y 607.847,Z 355.325,A -85,B 0,C 180,E1 27690.972,E2 27690.972} C_VEL
LIN {X 0,Y 607.905,Z 355.324,A -85,B 0,C 180,E1 27688.021,E2 27688.021} C_VEL
LIN {X 0,Y 607.837,Z 355.327,A -85,B 0,C 180,E1 27684.965,E2 27684.965} C_VEL
LIN {X 0,Y 607.872,Z 355.327,A -85,B 0,C 180,E1 27682.036,E2 27682.036} C_VEL
LIN {X 0,Y 607.831,Z 355.328,A -85,B 0,C 180,E1 27678.887,E2 27678.887} C_VEL
LIN {X 0,Y 607.856,Z 355.328,A -85,B 0,C 180,E1 27676.041,E2 27676.041} C_VEL
LIN {X 0,Y 607.843,Z 355.325,A -85,B 0,C 180,E1 27672.795,E2 27672.795} C_VEL
LIN {X 0,Y 607.856,Z 355.316,A -85,B 0,C 180,E1 27670.029,E2 27670.029} C_VEL
LIN {X 0,Y 607.885,Z 355.946,A -85,B 0,C 180,E1 27669.739,E2 27669.739} C_VEL
LIN {X 0,Y 607.918,Z 390.475,A -85,B 0,C 180,E1 27667.402,E2 27667.402} C_VEL
LIN {X 0,Y 607.916,Z 399.223,A -85,B 0,C 180,E1 27667.246,E2 27667.246} C_VEL
LIN {X 0,Y 607.916,Z 605.62,A -85,B 0,C 180,E1 27664.302,E2 27664.302} C_VEL
LIN {X 0,Y 607.913,Z 739.011,A -85,B 0,C 180,E1 27662.426,E2 27662.426} C_VEL
LIN {X 0,Y 607.915,Z 761.995,A -85,B 0,C 180,E1 27661.932,E2 27661.932} C_VEL
LIN {X 0,Y 607.917,Z 780.55,A -85,B 0,C 180,E1 27661.394,E2 27661.394} C_VEL
LIN {X 0,Y 607.912,Z 801.881,A -85,B 0,C 180,E1 27660.63,E2 27660.63} C_VEL
LIN {X 0,Y 607.919,Z 822.107,A -85,B 0,C 180,E1 27659.726,E2 27659.726} C_VEL
LIN {X 0,Y 607.916,Z 842.726,A -85,B 0,C 180,E1 27658.651,E2 27658.651} C_VEL
LIN {X 0,Y 607.917,Z 862.532,A -85,B 0,C 180,E1 27657.423,E2 27657.423} C_VEL
LIN {X 0,Y 607.912,Z 881.932,A -85,B 0,C 180,E1 27656.051,E2 27656.051} C_VEL
LIN {X 0,Y 607.91,Z 900.181,A -85,B 0,C 180,E1 27654.558,E2 27654.558} C_VEL
LIN {X 0,Y 607.916,Z 918.576,A -85,B 0,C 180,E1 27652.842,E2 27652.842} C_VEL
LIN {X 0,Y 607.912,Z 934.857,A -85,B 0,C 180,E1 27651.115,E2 27651.115} C_VEL
LIN {X 0,Y 607.91,Z 950.073,A -85,B 0,C 180,E1 27649.252,E2 27649.252} C_VEL
LIN {X 0,Y 607.911,Z 964.502,A -85,B 0,C 180,E1 27647.223,E2 27647.223} C_VEL
LIN {X 0,Y 607.9,Z 976.021,A -85,B 0,C 180,E1 27645.358,E2 27645.358} C_VEL
LIN {X 0,Y 607.885,Z 986.743,A -85,B 0,C 180,E1 27643.316,E2 27643.316} C_VEL
LIN {X 0,Y 607.907,Z 995.299,A -85,B 0,C 180,E1 27641.401,E2 27641.401} C_VEL
LIN {X 0,Y 607.896,Z 1003.029,A -85,B 0,C 180,E1 27639.278,E2 27639.278} C_VEL
LIN {X 0,Y 607.888,Z 1008.583,A -85,B 0,C 180,E1 27637.374,E2 27637.374} C_VEL
LIN {X 0,Y 607.911,Z 1013.315,A -85,B 0,C 180,E1 27635.193,E2 27635.193} C_VEL
LIN {X 0,Y 607.882,Z 1016.063,A -85,B 0,C 180,E1 27633.303,E2 27633.303} C_VEL
LIN {X 0,Y 607.905,Z 1017.738,A -85,B 0,C 180,E1 27631.134,E2 27631.134} C_VEL
LIN {X 0,Y 607.886,Z 1017.806,A -85,B 0,C 180,E1 27629.155,E2 27629.155} C_VEL
LIN {X 0,Y 607.884,Z 1016.408,A -85,B 0,C 180,E1 27626.986,E2 27626.986} C_VEL
LIN {X 0,Y 607.907,Z 1013.643,A -85,B 0,C 180,E1 27625.002,E2 27625.002} C_VEL
LIN {X 0,Y 607.882,Z 1009.109,A -85,B 0,C 180,E1 27622.822,E2 27622.822} C_VEL
LIN {X 0,Y 607.904,Z 1003.353,A -85,B 0,C 180,E1 27620.823,E2 27620.823} C_VEL
LIN {X 0,Y 607.898,Z 995.798,A -85,B 0,C 180,E1 27618.716,E2 27618.716} C_VEL
LIN {X 0,Y 607.889,Z 987.235,A -85,B 0,C 180,E1 27616.787,E2 27616.787} C_VEL
LIN {X 0,Y 607.911,Z 977.201,A -85,B 0,C 180,E1 27614.844,E2 27614.844} C_VEL
LIN {X 0,Y 607.908,Z 965.052,A -85,B 0,C 180,E1 27612.861,E2 27612.861} C_VEL
LIN {X 0,Y 607.906,Z 951.246,A -85,B 0,C 180,E1 27610.898,E2 27610.898} C_VEL
LIN {X 0,Y 607.91,Z 936.613,A -85,B 0,C 180,E1 27609.093,E2 27609.093} C_VEL
LIN {X 0,Y 607.914,Z 920.209,A -85,B 0,C 180,E1 27607.323,E2 27607.323} C_VEL
LIN {X 0,Y 607.905,Z 902.853,A -85,B 0,C 180,E1 27605.67,E2 27605.67} C_VEL
LIN {X 0,Y 607.908,Z 884.66,A -85,B 0,C 180,E1 27604.164,E2 27604.164} C_VEL
LIN {X 0,Y 607.913,Z 864.234,A -85,B 0,C 180,E1 27602.689,E2 27602.689} C_VEL
LIN {X 0,Y 607.916,Z 844.867,A -85,B 0,C 180,E1 27601.476,E2 27601.476} C_VEL
LIN {X 0,Y 607.918,Z 824.394,A -85,B 0,C 180,E1 27600.385,E2 27600.385} C_VEL
LIN {X 0,Y 607.914,Z 805.451,A -85,B 0,C 180,E1 27599.523,E2 27599.523} C_VEL
LIN {X 0,Y 607.915,Z 783.176,A -85,B 0,C 180,E1 27598.69,E2 27598.69} C_VEL
LIN {X 0,Y 607.913,Z 764.577,A -85,B 0,C 180,E1 27598.137,E2 27598.137} C_VEL
LIN {X 0,Y 607.91,Z 742.837,A -85,B 0,C 180,E1 27597.636,E2 27597.636} C_VEL
LIN {X 0,Y 607.915,Z 700.776,A -85,B 0,C 180,E1 27597.021,E2 27597.021} C_VEL
LIN {X 0,Y 607.914,Z 491.097,A -85,B 0,C 180,E1 27594.078,E2 27594.078} C_VEL
LIN {X 0,Y 607.918,Z 390.776,A -85,B 0,C 180,E1 27592.619,E2 27592.619} C_VEL
LIN {X 0,Y 607.887,Z 355.822,A -85,B 0,C 180,E1 27590.253,E2 27590.253} C_VEL
LIN {X 0,Y 607.858,Z 355.316,A -85,B 0,C 180,E1 27589.978,E2 27589.978} C_VEL
LIN {X 0,Y 607.846,Z 355.324,A -85,B 0,C 180,E1 27587.191,E2 27587.191} C_VEL
LIN {X 0,Y 607.879,Z 355.326,A -85,B 0,C 180,E1 27584.052,E2 27584.052} C_VEL
LIN {X 0,Y 607.837,Z 355.326,A -85,B 0,C 180,E1 27581.145,E2 27581.145} C_VEL
LIN {X 0,Y 607.896,Z 355.328,A -85,B 0,C 180,E1 27578.022,E2 27578.022} C_VEL
LIN {X 0,Y 607.829,Z 355.326,A -85,B 0,C 180,E1 27575.151,E2 27575.151} C_VEL
LIN {X 0,Y 607.897,Z 355.326,A -85,B 0,C 180,E1 27572.202,E2 27572.202} C_VEL
LIN {X 0,Y 607.827,Z 355.327,A -85,B 0,C 180,E1 27569.137,E2 27569.137} C_VEL
LIN {X 0,Y 607.838,Z 355.327,A -85,B 0,C 180,E1 27566.473,E2 27566.473} C_VEL
LIN {X 0,Y 607.837,Z 355.327,A -85,B 0,C 180,E1 27563.15,E2 27563.15} C_VEL
LIN {X 0,Y 607.834,Z 355.327,A -85,B 0,C 180,E1 27560.409,E2 27560.409} C_VEL
LIN {X 0,Y 607.865,Z 355.326,A -85,B 0,C 180,E1 27557.222,E2 27557.222} C_VEL
LIN {X 0,Y 607.833,Z 355.326,A -85,B 0,C 180,E1 27554.352,E2 27554.352} C_VEL
LIN {X 0,Y 607.902,Z 355.325,A -85,B 0,C 180,E1 27551.287,E2 27551.287} C_VEL
LIN {X 0,Y 607.835,Z 355.326,A -85,B 0,C 180,E1 27548.323,E2 27548.323} C_VEL
LIN {X 0,Y 607.915,Z 355.327,A -85,B 0,C 180,E1 27545.284,E2 27545.284} C_VEL
LIN {X 0,Y 607.84,Z 355.325,A -85,B 0,C 180,E1 27542.262,E2 27542.262} C_VEL
LIN {X 0,Y 607.896,Z 355.327,A -85,B 0,C 180,E1 27539.34,E2 27539.34} C_VEL
LIN {X 0,Y 607.886,Z 355.323,A -85,B 0,C 180,E1 27536.669,E2 27536.669} C_VEL
LIN {X 0,Y 606.83,Z 355.455,A -85,B 0,C 180,E1 27535.943,E2 27535.943} C_VEL
LIN {X 0,Y 600.418,Z 356.253,A -85,B 0,C 180,E1 27533.906,E2 27533.906} C_VEL
LIN {X 0,Y 599.935,Z 356.316,A -85,B 0,C 180,E1 27533.376,E2 27533.376} C_VEL
LIN {X 0,Y 599.918,Z 356.313,A -85,B 0,C 180,E1 27530.115,E2 27530.115} C_VEL
LIN {X 0,Y 599.94,Z 356.315,A -85,B 0,C 180,E1 27527.193,E2 27527.193} C_VEL
LIN {X 0,Y 599.923,Z 356.312,A -85,B 0,C 180,E1 27523.938,E2 27523.938} C_VEL
LIN {X 0,Y 599.959,Z 356.315,A -85,B 0,C 180,E1 27520.881,E2 27520.881} C_VEL
LIN {X 0,Y 599.923,Z 356.311,A -85,B 0,C 180,E1 27517.653,E2 27517.653} C_VEL
LIN {X 0,Y 599.973,Z 356.316,A -85,B 0,C 180,E1 27514.576,E2 27514.576} C_VEL
LIN {X 0,Y 599.923,Z 356.311,A -85,B 0,C 180,E1 27511.423,E2 27511.423} C_VEL
LIN {X 0,Y 599.978,Z 356.315,A -85,B 0,C 180,E1 27508.335,E2 27508.335} C_VEL
LIN {X 0,Y 599.927,Z 356.311,A -85,B 0,C 180,E1 27505.242,E2 27505.242} C_VEL
LIN {X 0,Y 599.977,Z 356.314,A -85,B 0,C 180,E1 27502.17,E2 27502.17} C_VEL
LIN {X 0,Y 599.931,Z 356.311,A -85,B 0,C 180,E1 27499.017,E2 27499.017} C_VEL
LIN {X 0,Y 599.972,Z 356.312,A -85,B 0,C 180,E1 27495.845,E2 27495.845} C_VEL
LIN {X 0,Y 599.934,Z 356.311,A -85,B 0,C 180,E1 27492.694,E2 27492.694} C_VEL
LIN {X 0,Y 599.972,Z 356.312,A -85,B 0,C 180,E1 27489.652,E2 27489.652} C_VEL
LIN {X 0,Y 599.937,Z 356.312,A -85,B 0,C 180,E1 27486.506,E2 27486.506} C_VEL
LIN {X 0,Y 599.971,Z 356.309,A -85,B 0,C 180,E1 27483.359,E2 27483.359} C_VEL
LIN {X 0,Y 599.943,Z 356.312,A -85,B 0,C 180,E1 27480.215,E2 27480.215} C_VEL
LIN {X 0,Y 599.974,Z 356.307,A -85,B 0,C 180,E1 27476.927,E2 27476.927} C_VEL
LIN {X 0,Y 599.968,Z 356.314,A -85,B 0,C 180,E1 27473.676,E2 27473.676} C_VEL
LIN {X 0,Y 599.955,Z 356.307,A -85,B 0,C 180,E1 27470.38,E2 27470.38} C_VEL
LIN {X 0,Y 599.965,Z 356.308,A -85,B 0,C 180,E1 27467.152,E2 27467.152} C_VEL
LIN {X 0,Y 599.95,Z 356.311,A -85,B 0,C 180,E1 27463.981,E2 27463.981} C_VEL
LIN {X 0,Y 599.958,Z 356.274,A -85,B 0,C 180,E1 27460.851,E2 27460.851} C_VEL
LIN {X 0,Y 599.982,Z 356.369,A -85,B 0,C 180,E1 27460.268,E2 27460.268} C_VEL
LIN {X 0,Y 601.073,Z 360.1,A -85,B 0,C 180,E1 27459.911,E2 27459.911} C_VEL
LIN {X 0,Y 601.401,Z 362.833,A -85,B 0,C 180,E1 27459.769,E2 27459.769} C_VEL
LIN {X 0,Y 601.351,Z 510.629,A -85,B 0,C 180,E1 27457.615,E2 27457.615} C_VEL
LIN {X 0,Y 601.149,Z 709.656,A -85,B 0,C 180,E1 27454.782,E2 27454.782} C_VEL
LIN {X 0,Y 601.07,Z 733.098,A -85,B 0,C 180,E1 27454.266,E2 27454.266} C_VEL
LIN {X 0,Y 600.999,Z 752.933,A -85,B 0,C 180,E1 27453.675,E2 27453.675} C_VEL
LIN {X 0,Y 600.875,Z 775.854,A -85,B 0,C 180,E1 27452.811,E2 27452.811} C_VEL
LIN {X 0,Y 600.791,Z 795.485,A -85,B 0,C 180,E1 27451.904,E2 27451.904} C_VEL
LIN {X 0,Y 600.65,Z 817.238,A -85,B 0,C 180,E1 27450.712,E2 27450.712} C_VEL
LIN {X 0,Y 600.547,Z 837.296,A -85,B 0,C 180,E1 27449.425,E2 27449.425} C_VEL
LIN {X 0,Y 600.416,Z 857.059,A -85,B 0,C 180,E1 27447.945,E2 27447.945} C_VEL
LIN {X 0,Y 600.293,Z 875.53,A -85,B 0,C 180,E1 27446.368,E2 27446.368} C_VEL
LIN {X 0,Y 600.211,Z 892.168,A -85,B 0,C 180,E1 27444.74,E2 27444.74} C_VEL
LIN {X 0,Y 600.118,Z 908.54,A -85,B 0,C 180,E1 27442.915,E2 27442.915} C_VEL
LIN {X 0,Y 600.057,Z 923.019,A -85,B 0,C 180,E1 27441.083,E2 27441.083} C_VEL
LIN {X 0,Y 600.004,Z 936.235,A -85,B 0,C 180,E1 27439.144,E2 27439.144} C_VEL
LIN {X 0,Y 599.973,Z 948.381,A -85,B 0,C 180,E1 27437.094,E2 27437.094} C_VEL
LIN {X 0,Y 599.942,Z 958.134,A -85,B 0,C 180,E1 27435.157,E2 27435.157} C_VEL
LIN {X 0,Y 599.903,Z 967.509,A -85,B 0,C 180,E1 27432.94,E2 27432.94} C_VEL
LIN {X 0,Y 599.923,Z 974.058,A -85,B 0,C 180,E1 27431.032,E2 27431.032} C_VEL
LIN {X 0,Y 599.903,Z 980.13,A -85,B 0,C 180,E1 27428.795,E2 27428.795} C_VEL
LIN {X 0,Y 599.888,Z 984.128,A -85,B 0,C 180,E1 27426.731,E2 27426.731} C_VEL
LIN {X 0,Y 599.91,Z 986.858,A -85,B 0,C 180,E1 27424.53,E2 27424.53} C_VEL
LIN {X 0,Y 599.889,Z 987.88,A -85,B 0,C 180,E1 27422.502,E2 27422.502} C_VEL
LIN {X 0,Y 599.886,Z 987.484,A -85,B 0,C 180,E1 27420.271,E2 27420.271} C_VEL
LIN {X 0,Y 599.904,Z 985.737,A -85,B 0,C 180,E1 27418.329,E2 27418.329} C_VEL
LIN {X 0,Y 599.883,Z 982.257,A -85,B 0,C 180,E1 27416.104,E2 27416.104} C_VEL
LIN {X 0,Y 599.91,Z 977.513,A -85,B 0,C 180,E1 27414.077,E2 27414.077} C_VEL
LIN {X 0,Y 599.916,Z 970.828,A -85,B 0,C 180,E1 27411.876,E2 27411.876} C_VEL
LIN {X 0,Y 599.912,Z 963.237,A -85,B 0,C 180,E1 27409.908,E2 27409.908} C_VEL
LIN {X 0,Y 599.956,Z 953.937,A -85,B 0,C 180,E1 27407.87,E2 27407.87} C_VEL
LIN {X 0,Y 599.987,Z 942.839,A -85,B 0,C 180,E1 27405.845,E2 27405.845} C_VEL
LIN {X 0,Y 600.031,Z 930.006,A -85,B 0,C 180,E1 27403.818,E2 27403.818} C_VEL
LIN {X 0,Y 600.082,Z 916.111,A -85,B 0,C 180,E1 27401.925,E2 27401.925} C_VEL
LIN {X 0,Y 600.175,Z 900.06,A -85,B 0,C 180,E1 27400.02,E2 27400.02} C_VEL
LIN {X 0,Y 600.274,Z 883.455,A -85,B 0,C 180,E1 27398.29,E2 27398.29} C_VEL
LIN {X 0,Y 600.348,Z 866.212,A -85,B 0,C 180,E1 27396.72,E2 27396.72} C_VEL
LIN {X 0,Y 600.481,Z 846.172,A -85,B 0,C 180,E1 27395.126,E2 27395.126} C_VEL
LIN {X 0,Y 600.607,Z 826.775,A -85,B 0,C 180,E1 27393.782,E2 27393.782} C_VEL
LIN {X 0,Y 600.72,Z 806.484,A -85,B 0,C 180,E1 27392.584,E2 27392.584} C_VEL
LIN {X 0,Y 600.852,Z 785.114,A -85,B 0,C 180,E1 27391.502,E2 27391.502} C_VEL
LIN {X 0,Y 600.94,Z 764.096,A -85,B 0,C 180,E1 27390.633,E2 27390.633} C_VEL
LIN {X 0,Y 601.044,Z 742.1,A -85,B 0,C 180,E1 27389.889,E2 27389.889} C_VEL
LIN {X 0,Y 601.113,Z 720.499,A -85,B 0,C 180,E1 27389.344,E2 27389.344} C_VEL
LIN {X 0,Y 601.17,Z 698.456,A -85,B 0,C 180,E1 27388.945,E2 27388.945} C_VEL
LIN {X 0,Y 601.404,Z 485.815,A -85,B 0,C 180,E1 27385.94,E2 27385.94} C_VEL
LIN {X 0,Y 601.375,Z 362.647,A -85,B 0,C 180,E1 27384.136,E2 27384.136} C_VEL
LIN {X 0,Y 601.099,Z 359.7,A -85,B 0,C 180,E1 27383.972,E2 27383.972} C_VEL
LIN {X 0,Y 599.982,Z 356.473,A -85,B 0,C 180,E1 27383.602,E2 27383.602} C_VEL
LIN {X 0,Y 599.972,Z 356.311,A -85,B 0,C 180,E1 27380.384,E2 27380.384} C_VEL
LIN {X 0,Y 599.946,Z 356.309,A -85,B 0,C 180,E1 27377.157,E2 27377.157} C_VEL
LIN {X 0,Y 599.968,Z 356.313,A -85,B 0,C 180,E1 27373.984,E2 27373.984} C_VEL
LIN {X 0,Y 599.95,Z 356.31,A -85,B 0,C 180,E1 27370.855,E2 27370.855} C_VEL
LIN {X 0,Y 599.961,Z 356.31,A -85,B 0,C 180,E1 27367.662,E2 27367.662} C_VEL
LIN {X 0,Y 599.959,Z 356.312,A -85,B 0,C 180,E1 27364.493,E2 27364.493} C_VEL
LIN {X 0,Y 599.964,Z 356.307,A -85,B 0,C 180,E1 27361.242,E2 27361.242} C_VEL
LIN {X 0,Y 599.965,Z 356.314,A -85,B 0,C 180,E1 27357.899,E2 27357.899} C_VEL
LIN {X 0,Y 599.971,Z 356.308,A -85,B 0,C 180,E1 27354.645,E2 27354.645} C_VEL
LIN {X 0,Y 599.943,Z 356.312,A -85,B 0,C 180,E1 27351.47,E2 27351.47} C_VEL
LIN {X 0,Y 599.972,Z 356.31,A -85,B 0,C 180,E1 27348.367,E2 27348.367} C_VEL
LIN {X 0,Y 599.933,Z 356.312,A -85,B 0,C 180,E1 27345.227,E2 27345.227} C_VEL
LIN {X 0,Y 599.976,Z 356.314,A -85,B 0,C 180,E1 27342.043,E2 27342.043} C_VEL
LIN {X 0,Y 599.926,Z 356.311,A -85,B 0,C 180,E1 27338.901,E2 27338.901} C_VEL
LIN {X 0,Y 599.961,Z 356.316,A -85,B 0,C 180,E1 27335.693,E2 27335.693} C_VEL
LIN {X 0,Y 599.918,Z 356.313,A -85,B 0,C 180,E1 27332.666,E2 27332.666} C_VEL
LIN {X 0,Y 599.937,Z 356.316,A -85,B 0,C 180,E1 27329.449,E2 27329.449} C_VEL
LIN {X 0,Y 599.904,Z 356.315,A -85,B 0,C 180,E1 27326.619,E2 27326.619} C_VEL
LIN {X 0,Y 599.943,Z 356.317,A -85,B 0,C 180,E1 27323.448,E2 27323.448} C_VEL
LIN {X 0,Y 599.89,Z 356.317,A -85,B 0,C 180,E1 27320.508,E2 27320.508} C_VEL
LIN {X 0,Y 599.953,Z 356.317,A -85,B 0,C 180,E1 27317.42,E2 27317.42} C_VEL
LIN {X 0,Y 599.894,Z 356.317,A -85,B 0,C 180,E1 27314.492,E2 27314.492} C_VEL
LIN {X 0,Y 599.978,Z 356.288,A -85,B 0,C 180,E1 27311.417,E2 27311.417} C_VEL
LIN {X 0,Y 599.938,Z 356.56,A -85,B 0,C 180,E1 27310.358,E2 27310.358} C_VEL
LIN {X 0,Y 601.27,Z 360.463,A -85,B 0,C 180,E1 27309.934,E2 27309.934} C_VEL
LIN {X 0,Y 601.279,Z 391.48,A -85,B 0,C 180,E1 27307.846,E2 27307.846} C_VEL
LIN {X 0,Y 601.544,Z 396.097,A -85,B 0,C 180,E1 27307.755,E2 27307.755} C_VEL
LIN {X 0,Y 601.308,Z 602.567,A -85,B 0,C 180,E1 27304.776,E2 27304.776} C_VEL
LIN {X 0,Y 601.147,Z 739.225,A -85,B 0,C 180,E1 27302.833,E2 27302.833} C_VEL
LIN {X 0,Y 601.067,Z 762.953,A -85,B 0,C 180,E1 27302.314,E2 27302.314} C_VEL
LIN {X 0,Y 601.001,Z 782.306,A -85,B 0,C 180,E1 27301.74,E2 27301.74} C_VEL
LIN {X 0,Y 600.876,Z 805.207,A -85,B 0,C 180,E1 27300.883,E2 27300.883} C_VEL
LIN {X 0,Y 600.793,Z 824.261,A -85,B 0,C 180,E1 27300.009,E2 27300.009} C_VEL
LIN {X 0,Y 600.656,Z 845.436,A -85,B 0,C 180,E1 27298.866,E2 27298.866} C_VEL
LIN {X 0,Y 600.556,Z 864.862,A -85,B 0,C 180,E1 27297.632,E2 27297.632} C_VEL
LIN {X 0,Y 600.418,Z 884.953,A -85,B 0,C 180,E1 27296.159,E2 27296.159} C_VEL
LIN {X 0,Y 600.324,Z 903.725,A -85,B 0,C 180,E1 27294.581,E2 27294.581} C_VEL
LIN {X 0,Y 600.228,Z 921.027,A -85,B 0,C 180,E1 27292.901,E2 27292.901} C_VEL
LIN {X 0,Y 600.13,Z 938.266,A -85,B 0,C 180,E1 27290.992,E2 27290.992} C_VEL
LIN {X 0,Y 600.066,Z 952.978,A -85,B 0,C 180,E1 27289.134,E2 27289.134} C_VEL
LIN {X 0,Y 600.009,Z 966.432,A -85,B 0,C 180,E1 27287.157,E2 27287.157} C_VEL
LIN {X 0,Y 599.973,Z 978.737,A -85,B 0,C 180,E1 27285.071,E2 27285.071} C_VEL
LIN {X 0,Y 599.925,Z 988.136,A -85,B 0,C 180,E1 27283.201,E2 27283.201} C_VEL
LIN {X 0,Y 599.905,Z 997.258,A -85,B 0,C 180,E1 27281.053,E2 27281.053} C_VEL
LIN {X 0,Y 599.919,Z 1003.944,A -85,B 0,C 180,E1 27279.113,E2 27279.113} C_VEL
LIN {X 0,Y 599.885,Z 1009.801,A -85,B 0,C 180,E1 27276.991,E2 27276.991} C_VEL
LIN {X 0,Y 599.906,Z 1013.793,A -85,B 0,C 180,E1 27274.975,E2 27274.975} C_VEL
LIN {X 0,Y 599.892,Z 1016.627,A -85,B 0,C 180,E1 27272.869,E2 27272.869} C_VEL
LIN {X 0,Y 599.884,Z 1017.827,A -85,B 0,C 180,E1 27270.767,E2 27270.767} C_VEL
LIN {X 0,Y 599.915,Z 1017.694,A -85,B 0,C 180,E1 27268.666,E2 27268.666} C_VEL
LIN {X 0,Y 599.886,Z 1015.957,A -85,B 0,C 180,E1 27266.563,E2 27266.563} C_VEL
LIN {X 0,Y 599.9,Z 1013.007,A -85,B 0,C 180,E1 27264.552,E2 27264.552} C_VEL
LIN {X 0,Y 599.914,Z 1008.088,A -85,B 0,C 180,E1 27262.341,E2 27262.341} C_VEL
LIN {X 0,Y 599.893,Z 1002.438,A -85,B 0,C 180,E1 27260.409,E2 27260.409} C_VEL
LIN {X 0,Y 599.929,Z 994.163,A -85,B 0,C 180,E1 27258.174,E2 27258.174} C_VEL
LIN {X 0,Y 599.935,Z 985.845,A -85,B 0,C 180,E1 27256.314,E2 27256.314} C_VEL
LIN {X 0,Y 599.967,Z 974.316,A -85,B 0,C 180,E1 27254.142,E2 27254.142} C_VEL
LIN {X 0,Y 600.009,Z 962.614,A -85,B 0,C 180,E1 27252.248,E2 27252.248} C_VEL
LIN {X 0,Y 600.079,Z 948.551,A -85,B 0,C 180,E1 27250.288,E2 27250.288} C_VEL
LIN {X 0,Y 600.164,Z 933.092,A -85,B 0,C 180,E1 27248.401,E2 27248.401} C_VEL
LIN {X 0,Y 600.237,Z 917.116,A -85,B 0,C 180,E1 27246.699,E2 27246.699} C_VEL
LIN {X 0,Y 600.347,Z 899.258,A -85,B 0,C 180,E1 27245.031,E2 27245.031} C_VEL
LIN {X 0,Y 600.47,Z 880.657,A -85,B 0,C 180,E1 27243.501,E2 27243.501} C_VEL
LIN {X 0,Y 600.566,Z 861.027,A -85,B 0,C 180,E1 27242.111,E2 27242.111} C_VEL
LIN {X 0,Y 600.708,Z 839.876,A -85,B 0,C 180,E1 27240.816,E2 27240.816} C_VEL
LIN {X 0,Y 600.801,Z 819.813,A -85,B 0,C 180,E1 27239.772,E2 27239.772} C_VEL
LIN {X 0,Y 600.932,Z 797.653,A -85,B 0,C 180,E1 27238.813,E2 27238.813} C_VEL
LIN {X 0,Y 601.009,Z 777.904,A -85,B 0,C 180,E1 27238.117,E2 27238.117} C_VEL
LIN {X 0,Y 601.106,Z 754.863,A -85,B 0,C 180,E1 27237.485,E2 27237.485} C_VEL
LIN {X 0,Y 601.152,Z 735.147,A -85,B 0,C 180,E1 27237.099,E2 27237.099} C_VEL
LIN {X 0,Y 601.402,Z 510.443,A -85,B 0,C 180,E1 27233.908,E2 27233.908} C_VEL
LIN {X 0,Y 601.373,Z 391.969,A -85,B 0,C 180,E1 27232.171,E2 27232.171} C_VEL
LIN {X 0,Y 601.163,Z 388.321,A -85,B 0,C 180,E1 27231.965,E2 27231.965} C_VEL
LIN {X 0,Y 601.106,Z 359.613,A -85,B 0,C 180,E1 27229.994,E2 27229.994} C_VEL
LIN {X 0,Y 599.929,Z 356.499,A -85,B 0,C 180,E1 27229.633,E2 27229.633} C_VEL
LIN {X 0,Y 599.918,Z 356.311,A -85,B 0,C 180,E1 27227.025,E2 27227.025} C_VEL
LIN {X 0,Y 599.911,Z 356.313,A -85,B 0,C 180,E1 27223.762,E2 27223.762} C_VEL
LIN {X 0,Y 599.905,Z 356.316,A -85,B 0,C 180,E1 27220.981,E2 27220.981} C_VEL
LIN {X 0,Y 599.914,Z 356.317,A -85,B 0,C 180,E1 27217.666,E2 27217.666} C_VEL
LIN {X 0,Y 599.894,Z 356.313,A -85,B 0,C 180,E1 27214.921,E2 27214.921} C_VEL
LIN {X 0,Y 599.943,Z 356.315,A -85,B 0,C 180,E1 27211.778,E2 27211.778} C_VEL
LIN {X 0,Y 599.885,Z 356.316,A -85,B 0,C 180,E1 27208.904,E2 27208.904} C_VEL
LIN {X 0,Y 599.969,Z 356.317,A -85,B 0,C 180,E1 27205.864,E2 27205.864} C_VEL
LIN {X 0,Y 599.886,Z 356.316,A -85,B 0,C 180,E1 27202.835,E2 27202.835} C_VEL
LIN {X 0,Y 599.951,Z 356.316,A -85,B 0,C 180,E1 27199.875,E2 27199.875} C_VEL
LIN {X 0,Y 599.892,Z 356.316,A -85,B 0,C 180,E1 27196.758,E2 27196.758} C_VEL
LIN {X 0,Y 599.93,Z 356.316,A -85,B 0,C 180,E1 27193.886,E2 27193.886} C_VEL
LIN {X 0,Y 599.904,Z 356.315,A -85,B 0,C 180,E1 27190.758,E2 27190.758} C_VEL
LIN {X 0,Y 599.912,Z 356.315,A -85,B 0,C 180,E1 27187.951,E2 27187.951} C_VEL
LIN {X 0,Y 599.911,Z 356.314,A -85,B 0,C 180,E1 27184.588,E2 27184.588} C_VEL
LIN {X 0,Y 599.92,Z 356.315,A -85,B 0,C 180,E1 27181.719,E2 27181.719} C_VEL
LIN {X 0,Y 599.92,Z 356.313,A -85,B 0,C 180,E1 27178.472,E2 27178.472} C_VEL
LIN {X 0,Y 599.919,Z 356.315,A -85,B 0,C 180,E1 27175.603,E2 27175.603} C_VEL
LIN {X 0,Y 599.935,Z 356.316,A -85,B 0,C 180,E1 27173.376,E2 27173.376} C_VEL
LIN {X 0,Y 599,Z 356.439,A -85,B 0,C 180,E1 27172.641,E2 27172.641} C_VEL
LIN {X 0,Y 592.435,Z 357.25,A -85,B 0,C 180,E1 27170.523,E2 27170.523} C_VEL
LIN {X 0,Y 591.976,Z 357.302,A -85,B 0,C 180,E1 27170.039,E2 27170.039} C_VEL
LIN {X 0,Y 592.022,Z 357.305,A -85,B 0,C 180,E1 27167.007,E2 27167.007} C_VEL
LIN {X 0,Y 591.979,Z 357.302,A -85,B 0,C 180,E1 27163.818,E2 27163.818} C_VEL
LIN {X 0,Y 592.034,Z 357.305,A -85,B 0,C 180,E1 27160.731,E2 27160.731} C_VEL
LIN {X 0,Y 591.981,Z 357.301,A -85,B 0,C 180,E1 27157.56,E2 27157.56} C_VEL
LIN {X 0,Y 592.036,Z 357.304,A -85,B 0,C 180,E1 27154.49,E2 27154.49} C_VEL
LIN {X 0,Y 591.983,Z 357.3,A -85,B 0,C 180,E1 27151.335,E2 27151.335} C_VEL
LIN {X 0,Y 592.039,Z 357.303,A -85,B 0,C 180,E1 27148.316,E2 27148.316} C_VEL
LIN {X 0,Y 591.987,Z 357.3,A -85,B 0,C 180,E1 27145.161,E2 27145.161} C_VEL
LIN {X 0,Y 592.036,Z 357.301,A -85,B 0,C 180,E1 27142.056,E2 27142.056} C_VEL
LIN {X 0,Y 591.991,Z 357.3,A -85,B 0,C 180,E1 27138.927,E2 27138.927} C_VEL
LIN {X 0,Y 592.034,Z 357.299,A -85,B 0,C 180,E1 27135.725,E2 27135.725} C_VEL
LIN {X 0,Y 591.997,Z 357.301,A -85,B 0,C 180,E1 27132.575,E2 27132.575} C_VEL
LIN {X 0,Y 592.035,Z 357.296,A -85,B 0,C 180,E1 27129.331,E2 27129.331} C_VEL
LIN {X 0,Y 592.016,Z 357.304,A -85,B 0,C 180,E1 27126.111,E2 27126.111} C_VEL
LIN {X 0,Y 592.011,Z 357.296,A -85,B 0,C 180,E1 27122.745,E2 27122.745} C_VEL
LIN {X 0,Y 592.034,Z 357.3,A -85,B 0,C 180,E1 27119.543,E2 27119.543} C_VEL
LIN {X 0,Y 592.005,Z 357.3,A -85,B 0,C 180,E1 27116.367,E2 27116.367} C_VEL
LIN {X 0,Y 592.029,Z 357.301,A -85,B 0,C 180,E1 27113.169,E2 27113.169} C_VEL
LIN {X 0,Y 592.007,Z 357.299,A -85,B 0,C 180,E1 27110.047,E2 27110.047} C_VEL
LIN {X 0,Y 592.025,Z 357.291,A -85,B 0,C 180,E1 27106.883,E2 27106.883} C_VEL
LIN {X 0,Y 592.015,Z 357.302,A -85,B 0,C 180,E1 27103.673,E2 27103.673} C_VEL
LIN {X 0,Y 592.036,Z 357.386,A -85,B 0,C 180,E1 27100.801,E2 27100.801} C_VEL
LIN {X 0,Y 593.91,Z 362.11,A -85,B 0,C 180,E1 27100.343,E2 27100.343} C_VEL
LIN {X 0,Y 595.165,Z 365.099,A -85,B 0,C 180,E1 27100.202,E2 27100.202} C_VEL
LIN {X 0,Y 594.766,Z 557.471,A -85,B 0,C 180,E1 27097.389,E2 27097.389} C_VEL
LIN {X 0,Y 594.416,Z 709.835,A -85,B 0,C 180,E1 27095.199,E2 27095.199} C_VEL
LIN {X 0,Y 594.254,Z 733.404,A -85,B 0,C 180,E1 27094.675,E2 27094.675} C_VEL
LIN {X 0,Y 594.11,Z 753.87,A -85,B 0,C 180,E1 27094.056,E2 27094.056} C_VEL
LIN {X 0,Y 593.861,Z 776.625,A -85,B 0,C 180,E1 27093.182,E2 27093.182} C_VEL
LIN {X 0,Y 593.676,Z 798.14,A -85,B 0,C 180,E1 27092.169,E2 27092.169} C_VEL
LIN {X 0,Y 593.394,Z 819.424,A -85,B 0,C 180,E1 27090.962,E2 27090.962} C_VEL
LIN {X 0,Y 593.162,Z 839.911,A -85,B 0,C 180,E1 27089.611,E2 27089.611} C_VEL
LIN {X 0,Y 592.923,Z 859.35,A -85,B 0,C 180,E1 27088.113,E2 27088.113} C_VEL
LIN {X 0,Y 592.672,Z 878.493,A -85,B 0,C 180,E1 27086.418,E2 27086.418} C_VEL
LIN {X 0,Y 592.497,Z 895.766,A -85,B 0,C 180,E1 27084.672,E2 27084.672} C_VEL
LIN {X 0,Y 592.334,Z 911.685,A -85,B 0,C 180,E1 27082.822,E2 27082.822} C_VEL
LIN {X 0,Y 592.181,Z 926.374,A -85,B 0,C 180,E1 27080.865,E2 27080.865} C_VEL
LIN {X 0,Y 592.087,Z 939.547,A -85,B 0,C 180,E1 27078.855,E2 27078.855} C_VEL
LIN {X 0,Y 592.006,Z 950.904,A -85,B 0,C 180,E1 27076.818,E2 27076.818} C_VEL
LIN {X 0,Y 591.975,Z 960.95,A -85,B 0,C 180,E1 27074.72,E2 27074.72} C_VEL
LIN {X 0,Y 591.921,Z 968.91,A -85,B 0,C 180,E1 27072.702,E2 27072.702} C_VEL
LIN {X 0,Y 591.9,Z 975.886,A -85,B 0,C 180,E1 27070.56,E2 27070.56} C_VEL
LIN {X 0,Y 591.918,Z 980.967,A -85,B 0,C 180,E1 27068.495,E2 27068.495} C_VEL
LIN {X 0,Y 591.885,Z 984.946,A -85,B 0,C 180,E1 27066.29,E2 27066.29} C_VEL
LIN {X 0,Y 591.889,Z 987.14,A -85,B 0,C 180,E1 27064.16,E2 27064.16} C_VEL
LIN {X 0,Y 591.909,Z 987.997,A -85,B 0,C 180,E1 27061.99,E2 27061.99} C_VEL
LIN {X 0,Y 591.885,Z 987.226,A -85,B 0,C 180,E1 27059.873,E2 27059.873} C_VEL
LIN {X 0,Y 591.897,Z 985.197,A -85,B 0,C 180,E1 27057.813,E2 27057.813} C_VEL
LIN {X 0,Y 591.912,Z 981.219,A -85,B 0,C 180,E1 27055.534,E2 27055.534} C_VEL
LIN {X 0,Y 591.894,Z 976.324,A -85,B 0,C 180,E1 27053.513,E2 27053.513} C_VEL
LIN {X 0,Y 591.931,Z 969.232,A -85,B 0,C 180,E1 27051.297,E2 27051.297} C_VEL
LIN {X 0,Y 591.962,Z 961.436,A -85,B 0,C 180,E1 27049.307,E2 27049.307} C_VEL
LIN {X 0,Y 592,Z 951.653,A -85,B 0,C 180,E1 27047.236,E2 27047.236} C_VEL
LIN {X 0,Y 592.076,Z 940.597,A -85,B 0,C 180,E1 27045.233,E2 27045.233} C_VEL
LIN {X 0,Y 592.186,Z 927.972,A -85,B 0,C 180,E1 27043.275,E2 27043.275} C_VEL
LIN {X 0,Y 592.333,Z 913.434,A -85,B 0,C 180,E1 27041.301,E2 27041.301} C_VEL
LIN {X 0,Y 592.472,Z 897.491,A -85,B 0,C 180,E1 27039.431,E2 27039.431} C_VEL
LIN {X 0,Y 592.669,Z 880.056,A -85,B 0,C 180,E1 27037.641,E2 27037.641} C_VEL
LIN {X 0,Y 592.91,Z 861.696,A -85,B 0,C 180,E1 27035.988,E2 27035.988} C_VEL
LIN {X 0,Y 593.099,Z 842.666,A -85,B 0,C 180,E1 27034.503,E2 27034.503} C_VEL
LIN {X 0,Y 593.38,Z 821.734,A -85,B 0,C 180,E1 27033.09,E2 27033.09} C_VEL
LIN {X 0,Y 593.63,Z 800.664,A -85,B 0,C 180,E1 27031.873,E2 27031.873} C_VEL
LIN {X 0,Y 593.85,Z 778.928,A -85,B 0,C 180,E1 27030.829,E2 27030.829} C_VEL
LIN {X 0,Y 594.067,Z 757.974,A -85,B 0,C 180,E1 27029.992,E2 27029.992} C_VEL
LIN {X 0,Y 594.247,Z 735.854,A -85,B 0,C 180,E1 27029.303,E2 27029.303} C_VEL
LIN {X 0,Y 594.382,Z 713.433,A -85,B 0,C 180,E1 27028.774,E2 27028.774} C_VEL
LIN {X 0,Y 594.505,Z 674.523,A -85,B 0,C 180,E1 27028.186,E2 27028.186} C_VEL
LIN {X 0,Y 594.978,Z 464.25,A -85,B 0,C 180,E1 27025.172,E2 27025.172} C_VEL
LIN {X 0,Y 595.035,Z 364.461,A -85,B 0,C 180,E1 27023.688,E2 27023.688} C_VEL
LIN {X 0,Y 593.44,Z 360.972,A -85,B 0,C 180,E1 27023.483,E2 27023.483} C_VEL
LIN {X 0,Y 592.035,Z 357.58,A -85,B 0,C 180,E1 27023.094,E2 27023.094} C_VEL
LIN {X 0,Y 592.034,Z 357.301,A -85,B 0,C 180,E1 27021.707,E2 27021.707} C_VEL
LIN {X 0,Y 592.025,Z 357.289,A -85,B 0,C 180,E1 27018.411,E2 27018.411} C_VEL
LIN {X 0,Y 592.013,Z 357.297,A -85,B 0,C 180,E1 27015.176,E2 27015.176} C_VEL
LIN {X 0,Y 592.029,Z 357.303,A -85,B 0,C 180,E1 27011.99,E2 27011.99} C_VEL
LIN {X 0,Y 592.014,Z 357.299,A -85,B 0,C 180,E1 27008.841,E2 27008.841} C_VEL
LIN {X 0,Y 592.02,Z 357.3,A -85,B 0,C 180,E1 27005.719,E2 27005.719} C_VEL
LIN {X 0,Y 592.021,Z 357.301,A -85,B 0,C 180,E1 27002.517,E2 27002.517} C_VEL
LIN {X 0,Y 592.017,Z 357.298,A -85,B 0,C 180,E1 26999.323,E2 26999.323} C_VEL
LIN {X 0,Y 592.033,Z 357.306,A -85,B 0,C 180,E1 26996.03,E2 26996.03} C_VEL
LIN {X 0,Y 592.036,Z 357.296,A -85,B 0,C 180,E1 26992.724,E2 26992.724} C_VEL
LIN {X 0,Y 592.003,Z 357.302,A -85,B 0,C 180,E1 26989.49,E2 26989.49} C_VEL
LIN {X 0,Y 592.035,Z 357.3,A -85,B 0,C 180,E1 26986.324,E2 26986.324} C_VEL
LIN {X 0,Y 591.991,Z 357.301,A -85,B 0,C 180,E1 26983.213,E2 26983.213} C_VEL
LIN {X 0,Y 592.039,Z 357.302,A -85,B 0,C 180,E1 26980.054,E2 26980.054} C_VEL
LIN {X 0,Y 591.981,Z 357.301,A -85,B 0,C 180,E1 26976.931,E2 26976.931} C_VEL
LIN {X 0,Y 592.03,Z 357.304,A -85,B 0,C 180,E1 26973.738,E2 26973.738} C_VEL
LIN {X 0,Y 591.97,Z 357.302,A -85,B 0,C 180,E1 26970.783,E2 26970.783} C_VEL
LIN {X 0,Y 592.022,Z 357.306,A -85,B 0,C 180,E1 26967.631,E2 26967.631} C_VEL
LIN {X 0,Y 591.957,Z 357.305,A -85,B 0,C 180,E1 26964.671,E2 26964.671} C_VEL
LIN {X 0,Y 592.024,Z 357.305,A -85,B 0,C 180,E1 26961.574,E2 26961.574} C_VEL
LIN {X 0,Y 591.949,Z 357.307,A -85,B 0,C 180,E1 26958.538,E2 26958.538} C_VEL
LIN {X 0,Y 592.015,Z 357.302,A -85,B 0,C 180,E1 26955.366,E2 26955.366} C_VEL
LIN {X 0,Y 591.96,Z 357.299,A -85,B 0,C 180,E1 26952.374,E2 26952.374} C_VEL
LIN {X 0,Y 592.022,Z 357.55,A -85,B 0,C 180,E1 26950.94,E2 26950.94} C_VEL
LIN {X 0,Y 593.372,Z 360.961,A -85,B 0,C 180,E1 26950.54,E2 26950.54} C_VEL
LIN {X 0,Y 594.657,Z 364.043,A -85,B 0,C 180,E1 26950.217,E2 26950.217} C_VEL
LIN {X 0,Y 594.554,Z 391.477,A -85,B 0,C 180,E1 26948.351,E2 26948.351} C_VEL
LIN {X 0,Y 595.213,Z 395.815,A -85,B 0,C 180,E1 26948.233,E2 26948.233} C_VEL
LIN {X 0,Y 594.733,Z 602.312,A -85,B 0,C 180,E1 26945.221,E2 26945.221} C_VEL
LIN {X 0,Y 594.413,Z 739.44,A -85,B 0,C 180,E1 26943.25,E2 26943.25} C_VEL
LIN {X 0,Y 594.251,Z 763.127,A -85,B 0,C 180,E1 26942.726,E2 26942.726} C_VEL
LIN {X 0,Y 594.113,Z 782.973,A -85,B 0,C 180,E1 26942.13,E2 26942.13} C_VEL
LIN {X 0,Y 593.861,Z 806.355,A -85,B 0,C 180,E1 26941.238,E2 26941.238} C_VEL
LIN {X 0,Y 593.682,Z 826.501,A -85,B 0,C 180,E1 26940.294,E2 26940.294} C_VEL
LIN {X 0,Y 593.399,Z 848.109,A -85,B 0,C 180,E1 26939.088,E2 26939.088} C_VEL
LIN {X 0,Y 593.193,Z 868.454,A -85,B 0,C 180,E1 26937.76,E2 26937.76} C_VEL
LIN {X 0,Y 592.93,Z 887.231,A -85,B 0,C 180,E1 26936.329,E2 26936.329} C_VEL
LIN {X 0,Y 592.699,Z 906.325,A -85,B 0,C 180,E1 26934.67,E2 26934.67} C_VEL
LIN {X 0,Y 592.538,Z 923.319,A -85,B 0,C 180,E1 26932.978,E2 26932.978} C_VEL
LIN {X 0,Y 592.352,Z 939.119,A -85,B 0,C 180,E1 26931.177,E2 26931.177} C_VEL
LIN {X 0,Y 592.226,Z 953.605,A -85,B 0,C 180,E1 26929.308,E2 26929.308} C_VEL
LIN {X 0,Y 592.121,Z 966.434,A -85,B 0,C 180,E1 26927.393,E2 26927.393} C_VEL
LIN {X 0,Y 592.03,Z 978.738,A -85,B 0,C 180,E1 26925.278,E2 26925.278} C_VEL
LIN {X 0,Y 591.962,Z 988.186,A -85,B 0,C 180,E1 26923.371,E2 26923.371} C_VEL
LIN {X 0,Y 591.927,Z 997.259,A -85,B 0,C 180,E1 26921.204,E2 26921.204} C_VEL
LIN {X 0,Y 591.918,Z 1003.945,A -85,B 0,C 180,E1 26919.237,E2 26919.237} C_VEL
LIN {X 0,Y 591.888,Z 1009.801,A -85,B 0,C 180,E1 26917.086,E2 26917.086} C_VEL
LIN {X 0,Y 591.909,Z 1013.793,A -85,B 0,C 180,E1 26915.042,E2 26915.042} C_VEL
LIN {X 0,Y 591.89,Z 1016.627,A -85,B 0,C 180,E1 26912.908,E2 26912.908} C_VEL
LIN {X 0,Y 591.884,Z 1017.827,A -85,B 0,C 180,E1 26910.777,E2 26910.777} C_VEL
LIN {X 0,Y 591.914,Z 1017.694,A -85,B 0,C 180,E1 26908.648,E2 26908.648} C_VEL
LIN {X 0,Y 591.888,Z 1015.957,A -85,B 0,C 180,E1 26906.517,E2 26906.517} C_VEL
LIN {X 0,Y 591.899,Z 1013.007,A -85,B 0,C 180,E1 26904.478,E2 26904.478} C_VEL
LIN {X 0,Y 591.925,Z 1008.089,A -85,B 0,C 180,E1 26902.237,E2 26902.237} C_VEL
LIN {X 0,Y 591.903,Z 1002.439,A -85,B 0,C 180,E1 26900.278,E2 26900.278} C_VEL
LIN {X 0,Y 591.952,Z 994.164,A -85,B 0,C 180,E1 26898.013,E2 26898.013} C_VEL
LIN {X 0,Y 591.986,Z 985.846,A -85,B 0,C 180,E1 26896.127,E2 26896.127} C_VEL
LIN {X 0,Y 592.052,Z 974.318,A -85,B 0,C 180,E1 26893.925,E2 26893.925} C_VEL
LIN {X 0,Y 592.133,Z 962.615,A -85,B 0,C 180,E1 26892.004,E2 26892.004} C_VEL
LIN {X 0,Y 592.253,Z 948.914,A -85,B 0,C 180,E1 26890.065,E2 26890.065} C_VEL
LIN {X 0,Y 592.42,Z 933.633,A -85,B 0,C 180,E1 26888.165,E2 26888.165} C_VEL
LIN {X 0,Y 592.568,Z 917.622,A -85,B 0,C 180,E1 26886.432,E2 26886.432} C_VEL
LIN {X 0,Y 592.794,Z 899.328,A -85,B 0,C 180,E1 26884.697,E2 26884.697} C_VEL
LIN {X 0,Y 593.043,Z 880.658,A -85,B 0,C 180,E1 26883.142,E2 26883.142} C_VEL
LIN {X 0,Y 593.241,Z 861.03,A -85,B 0,C 180,E1 26881.736,E2 26881.736} C_VEL
LIN {X 0,Y 593.526,Z 839.88,A -85,B 0,C 180,E1 26880.428,E2 26880.428} C_VEL
LIN {X 0,Y 593.716,Z 819.925,A -85,B 0,C 180,E1 26879.379,E2 26879.379} C_VEL
LIN {X 0,Y 593.98,Z 797.58,A -85,B 0,C 180,E1 26878.403,E2 26878.403} C_VEL
LIN {X 0,Y 594.136,Z 777.261,A -85,B 0,C 180,E1 26877.683,E2 26877.683} C_VEL
LIN {X 0,Y 594.331,Z 753.457,A -85,B 0,C 180,E1 26877.037,E2 26877.037} C_VEL
LIN {X 0,Y 594.427,Z 733.864,A -85,B 0,C 180,E1 26876.657,E2 26876.657} C_VEL
LIN {X 0,Y 594.927,Z 512.688,A -85,B 0,C 180,E1 26873.485,E2 26873.485} C_VEL
LIN {X 0,Y 595.051,Z 393.776,A -85,B 0,C 180,E1 26871.724,E2 26871.724} C_VEL
LIN {X 0,Y 594.438,Z 390.12,A -85,B 0,C 180,E1 26871.579,E2 26871.579} C_VEL
LIN {X 0,Y 594.61,Z 363.854,A -85,B 0,C 180,E1 26869.766,E2 26869.766} C_VEL
LIN {X 0,Y 592.04,Z 357.671,A -85,B 0,C 180,E1 26869.091,E2 26869.091} C_VEL
LIN {X 0,Y 592.031,Z 357.265,A -85,B 0,C 180,E1 26868.422,E2 26868.422} C_VEL
LIN {X 0,Y 591.96,Z 357.306,A -85,B 0,C 180,E1 26865.366,E2 26865.366} C_VEL
LIN {X 0,Y 592.032,Z 357.303,A -85,B 0,C 180,E1 26862.234,E2 26862.234} C_VEL
LIN {X 0,Y 591.956,Z 357.301,A -85,B 0,C 180,E1 26859.176,E2 26859.176} C_VEL
LIN {X 0,Y 592.037,Z 357.3,A -85,B 0,C 180,E1 26856.114,E2 26856.114} C_VEL
LIN {X 0,Y 591.951,Z 357.306,A -85,B 0,C 180,E1 26853.064,E2 26853.064} C_VEL
LIN {X 0,Y 592.034,Z 357.3,A -85,B 0,C 180,E1 26849.969,E2 26849.969} C_VEL
LIN {X 0,Y 591.946,Z 357.306,A -85,B 0,C 180,E1 26846.905,E2 26846.905} C_VEL
LIN {X 0,Y 592.032,Z 357.305,A -85,B 0,C 180,E1 26843.805,E2 26843.805} C_VEL
LIN {X 0,Y 591.949,Z 357.305,A -85,B 0,C 180,E1 26840.775,E2 26840.775} C_VEL
LIN {X 0,Y 592.028,Z 357.305,A -85,B 0,C 180,E1 26837.697,E2 26837.697} C_VEL
LIN {X 0,Y 591.953,Z 357.304,A -85,B 0,C 180,E1 26834.576,E2 26834.576} C_VEL
LIN {X 0,Y 592.036,Z 357.304,A -85,B 0,C 180,E1 26831.495,E2 26831.495} C_VEL
LIN {X 0,Y 591.959,Z 357.303,A -85,B 0,C 180,E1 26828.45,E2 26828.45} C_VEL
LIN {X 0,Y 592.026,Z 357.305,A -85,B 0,C 180,E1 26825.427,E2 26825.427} C_VEL
LIN {X 0,Y 591.965,Z 357.302,A -85,B 0,C 180,E1 26822.323,E2 26822.323} C_VEL
LIN {X 0,Y 592.02,Z 357.305,A -85,B 0,C 180,E1 26819.322,E2 26819.322} C_VEL
LIN {X 0,Y 591.969,Z 357.302,A -85,B 0,C 180,E1 26816.126,E2 26816.126} C_VEL
LIN {X 0,Y 592.029,Z 357.305,A -85,B 0,C 180,E1 26813.113,E2 26813.113} C_VEL
LIN {X 0,Y 591.976,Z 357.302,A -85,B 0,C 180,E1 26810.039,E2 26810.039} C_VEL
LIN {X 0,Y 590.98,Z 357.432,A -85,B 0,C 180,E1 26809.294,E2 26809.294} C_VEL
LIN {X 0,Y 584.63,Z 358.23,A -85,B 0,C 180,E1 26807.201,E2 26807.201} C_VEL
LIN {X 0,Y 584.1,Z 358.29,A -85,B 0,C 180,E1 26806.657,E2 26806.657} C_VEL
LIN {X 0,Y 584.039,Z 358.292,A -85,B 0,C 180,E1 26803.489,E2 26803.489} C_VEL
LIN {X 0,Y 584.09,Z 358.288,A -85,B 0,C 180,E1 26800.29,E2 26800.29} C_VEL
LIN {X 0,Y 584.045,Z 358.291,A -85,B 0,C 180,E1 26797.238,E2 26797.238} C_VEL
LIN {X 0,Y 584.081,Z 358.288,A -85,B 0,C 180,E1 26793.979,E2 26793.979} C_VEL
LIN {X 0,Y 584.056,Z 358.291,A -85,B 0,C 180,E1 26790.909,E2 26790.909} C_VEL
LIN {X 0,Y 584.062,Z 358.288,A -85,B 0,C 180,E1 26787.552,E2 26787.552} C_VEL
LIN {X 0,Y 584.092,Z 358.293,A -85,B 0,C 180,E1 26784.393,E2 26784.393} C_VEL
LIN {X 0,Y 584.055,Z 358.288,A -85,B 0,C 180,E1 26781.155,E2 26781.155} C_VEL
LIN {X 0,Y 584.098,Z 358.291,A -85,B 0,C 180,E1 26777.974,E2 26777.974} C_VEL
LIN {X 0,Y 584.057,Z 358.289,A -85,B 0,C 180,E1 26774.848,E2 26774.848} C_VEL
LIN {X 0,Y 584.095,Z 358.29,A -85,B 0,C 180,E1 26771.724,E2 26771.724} C_VEL
LIN {X 0,Y 584.06,Z 358.29,A -85,B 0,C 180,E1 26768.524,E2 26768.524} C_VEL
LIN {X 0,Y 584.095,Z 358.284,A -85,B 0,C 180,E1 26765.26,E2 26765.26} C_VEL
LIN {X 0,Y 584.076,Z 358.291,A -85,B 0,C 180,E1 26762.046,E2 26762.046} C_VEL
LIN {X 0,Y 584.082,Z 358.282,A -85,B 0,C 180,E1 26758.748,E2 26758.748} C_VEL
LIN {X 0,Y 584.095,Z 358.287,A -85,B 0,C 180,E1 26755.442,E2 26755.442} C_VEL
LIN {X 0,Y 584.069,Z 358.289,A -85,B 0,C 180,E1 26752.226,E2 26752.226} C_VEL
LIN {X 0,Y 584.088,Z 358.289,A -85,B 0,C 180,E1 26749.08,E2 26749.08} C_VEL
LIN {X 0,Y 584.071,Z 358.282,A -85,B 0,C 180,E1 26745.893,E2 26745.893} C_VEL
LIN {X 0,Y 584.088,Z 358.264,A -85,B 0,C 180,E1 26742.644,E2 26742.644} C_VEL
LIN {X 0,Y 584.112,Z 358.427,A -85,B 0,C 180,E1 26741.349,E2 26741.349} C_VEL
LIN {X 0,Y 585.561,Z 361.962,A -85,B 0,C 180,E1 26740.996,E2 26740.996} C_VEL
LIN {X 0,Y 588.91,Z 367.877,A -85,B 0,C 180,E1 26740.641,E2 26740.641} C_VEL
LIN {X 0,Y 588.185,Z 574.74,A -85,B 0,C 180,E1 26737.592,E2 26737.592} C_VEL
LIN {X 0,Y 587.715,Z 710.191,A -85,B 0,C 180,E1 26735.623,E2 26735.623} C_VEL
LIN {X 0,Y 587.469,Z 733.712,A -85,B 0,C 180,E1 26735.093,E2 26735.093} C_VEL
LIN {X 0,Y 587.243,Z 754.789,A -85,B 0,C 180,E1 26734.446,E2 26734.446} C_VEL
LIN {X 0,Y 586.874,Z 777.394,A -85,B 0,C 180,E1 26733.562,E2 26733.562} C_VEL
LIN {X 0,Y 586.581,Z 798.82,A -85,B 0,C 180,E1 26732.537,E2 26732.537} C_VEL
LIN {X 0,Y 586.164,Z 820.045,A -85,B 0,C 180,E1 26731.316,E2 26731.316} C_VEL
LIN {X 0,Y 585.817,Z 840.438,A -85,B 0,C 180,E1 26729.948,E2 26729.948} C_VEL
LIN {X 0,Y 585.453,Z 859.851,A -85,B 0,C 180,E1 26728.431,E2 26728.431} C_VEL
LIN {X 0,Y 585.076,Z 878.926,A -85,B 0,C 180,E1 26726.715,E2 26726.715} C_VEL
LIN {X 0,Y 584.818,Z 895.694,A -85,B 0,C 180,E1 26724.995,E2 26724.995} C_VEL
LIN {X 0,Y 584.559,Z 911.621,A -85,B 0,C 180,E1 26723.121,E2 26723.121} C_VEL
LIN {X 0,Y 584.336,Z 926.313,A -85,B 0,C 180,E1 26721.139,E2 26721.139} C_VEL
LIN {X 0,Y 584.2,Z 939.211,A -85,B 0,C 180,E1 26719.146,E2 26719.146} C_VEL
LIN {X 0,Y 584.078,Z 950.835,A -85,B 0,C 180,E1 26717.038,E2 26717.038} C_VEL
LIN {X 0,Y 584.015,Z 960.885,A -85,B 0,C 180,E1 26714.914,E2 26714.914} C_VEL
LIN {X 0,Y 583.935,Z 968.971,A -85,B 0,C 180,E1 26712.835,E2 26712.835} C_VEL
LIN {X 0,Y 583.911,Z 975.964,A -85,B 0,C 180,E1 26710.65,E2 26710.65} C_VEL
LIN {X 0,Y 583.92,Z 981.143,A -85,B 0,C 180,E1 26708.502,E2 26708.502} C_VEL
LIN {X 0,Y 583.887,Z 985.062,A -85,B 0,C 180,E1 26706.268,E2 26706.268} C_VEL
LIN {X 0,Y 583.887,Z 987.199,A -85,B 0,C 180,E1 26704.106,E2 26704.106} C_VEL
LIN {X 0,Y 583.91,Z 987.995,A -85,B 0,C 180,E1 26701.905,E2 26701.905} C_VEL
LIN {X 0,Y 583.888,Z 987.176,A -85,B 0,C 180,E1 26699.769,E2 26699.769} C_VEL
LIN {X 0,Y 583.891,Z 984.983,A -85,B 0,C 180,E1 26697.587,E2 26697.587} C_VEL
LIN {X 0,Y 583.918,Z 981.027,A -85,B 0,C 180,E1 26695.353,E2 26695.353} C_VEL
LIN {X 0,Y 583.923,Z 975.508,A -85,B 0,C 180,E1 26693.097,E2 26693.097} C_VEL
LIN {X 0,Y 583.951,Z 968.49,A -85,B 0,C 180,E1 26690.94,E2 26690.94} C_VEL
LIN {X 0,Y 584.023,Z 959.704,A -85,B 0,C 180,E1 26688.728,E2 26688.728} C_VEL
LIN {X 0,Y 584.098,Z 949.695,A -85,B 0,C 180,E1 26686.65,E2 26686.65} C_VEL
LIN {X 0,Y 584.235,Z 937.1,A -85,B 0,C 180,E1 26684.424,E2 26684.424} C_VEL
LIN {X 0,Y 584.402,Z 923.651,A -85,B 0,C 180,E1 26682.385,E2 26682.385} C_VEL
LIN {X 0,Y 584.597,Z 908.523,A -85,B 0,C 180,E1 26680.408,E2 26680.408} C_VEL
LIN {X 0,Y 584.881,Z 891.647,A -85,B 0,C 180,E1 26678.482,E2 26678.482} C_VEL
LIN {X 0,Y 585.21,Z 874.063,A -85,B 0,C 180,E1 26676.727,E2 26676.727} C_VEL
LIN {X 0,Y 585.513,Z 855.428,A -85,B 0,C 180,E1 26675.116,E2 26675.116} C_VEL
LIN {X 0,Y 585.911,Z 834.832,A -85,B 0,C 180,E1 26673.567,E2 26673.567} C_VEL
LIN {X 0,Y 586.311,Z 813.681,A -85,B 0,C 180,E1 26672.203,E2 26672.203} C_VEL
LIN {X 0,Y 586.645,Z 792.158,A -85,B 0,C 180,E1 26671.036,E2 26671.036} C_VEL
LIN {X 0,Y 587.032,Z 770.414,A -85,B 0,C 180,E1 26670.05,E2 26670.05} C_VEL
LIN {X 0,Y 587.287,Z 748.712,A -85,B 0,C 180,E1 26669.262,E2 26669.262} C_VEL
LIN {X 0,Y 587.588,Z 725.248,A -85,B 0,C 180,E1 26668.602,E2 26668.602} C_VEL
LIN {X 0,Y 587.74,Z 703.248,A -85,B 0,C 180,E1 26668.17,E2 26668.17} C_VEL
LIN {X 0,Y 588.491,Z 485.386,A -85,B 0,C 180,E1 26665.015,E2 26665.015} C_VEL
LIN {X 0,Y 588.775,Z 367.303,A -85,B 0,C 180,E1 26663.25,E2 26663.25} C_VEL
LIN {X 0,Y 584.983,Z 361.13,A -85,B 0,C 180,E1 26662.83,E2 26662.83} C_VEL
LIN {X 0,Y 584.109,Z 358.478,A -85,B 0,C 180,E1 26662.521,E2 26662.521} C_VEL
LIN {X 0,Y 584.064,Z 358.268,A -85,B 0,C 180,E1 26659.189,E2 26659.189} C_VEL
LIN {X 0,Y 584.092,Z 358.29,A -85,B 0,C 180,E1 26655.998,E2 26655.998} C_VEL
LIN {X 0,Y 584.07,Z 358.291,A -85,B 0,C 180,E1 26652.758,E2 26652.758} C_VEL
LIN {X 0,Y 584.089,Z 358.287,A -85,B 0,C 180,E1 26649.558,E2 26649.558} C_VEL
LIN {X 0,Y 584.092,Z 358.293,A -85,B 0,C 180,E1 26646.29,E2 26646.29} C_VEL
LIN {X 0,Y 584.091,Z 358.285,A -85,B 0,C 180,E1 26642.944,E2 26642.944} C_VEL
LIN {X 0,Y 584.076,Z 358.291,A -85,B 0,C 180,E1 26639.706,E2 26639.706} C_VEL
LIN {X 0,Y 584.088,Z 358.288,A -85,B 0,C 180,E1 26636.467,E2 26636.467} C_VEL
LIN {X 0,Y 584.068,Z 358.289,A -85,B 0,C 180,E1 26633.316,E2 26633.316} C_VEL
LIN {X 0,Y 584.098,Z 358.293,A -85,B 0,C 180,E1 26630.044,E2 26630.044} C_VEL
LIN {X 0,Y 584.082,Z 358.287,A -85,B 0,C 180,E1 26626.739,E2 26626.739} C_VEL
LIN {X 0,Y 584.061,Z 358.292,A -85,B 0,C 180,E1 26623.472,E2 26623.472} C_VEL
LIN {X 0,Y 584.097,Z 358.288,A -85,B 0,C 180,E1 26620.293,E2 26620.293} C_VEL
LIN {X 0,Y 584.042,Z 358.291,A -85,B 0,C 180,E1 26617.08,E2 26617.08} C_VEL
LIN {X 0,Y 584.099,Z 358.293,A -85,B 0,C 180,E1 26613.901,E2 26613.901} C_VEL
LIN {X 0,Y 584.031,Z 358.291,A -85,B 0,C 180,E1 26610.797,E2 26610.797} C_VEL
LIN {X 0,Y 584.09,Z 358.293,A -85,B 0,C 180,E1 26607.718,E2 26607.718} C_VEL
LIN {X 0,Y 584.019,Z 358.295,A -85,B 0,C 180,E1 26604.752,E2 26604.752} C_VEL
LIN {X 0,Y 584.086,Z 358.294,A -85,B 0,C 180,E1 26601.582,E2 26601.582} C_VEL
LIN {X 0,Y 584.01,Z 358.297,A -85,B 0,C 180,E1 26598.582,E2 26598.582} C_VEL
LIN {X 0,Y 584.082,Z 358.288,A -85,B 0,C 180,E1 26595.41,E2 26595.41} C_VEL
LIN {X 0,Y 584.019,Z 358.274,A -85,B 0,C 180,E1 26592.42,E2 26592.42} C_VEL
LIN {X 0,Y 584.132,Z 358.539,A -85,B 0,C 180,E1 26591.541,E2 26591.541} C_VEL
LIN {X 0,Y 586.665,Z 364.805,A -85,B 0,C 180,E1 26590.825,E2 26590.825} C_VEL
LIN {X 0,Y 588.034,Z 367.765,A -85,B 0,C 180,E1 26590.498,E2 26590.498} C_VEL
LIN {X 0,Y 587.872,Z 391.473,A -85,B 0,C 180,E1 26588.868,E2 26588.868} C_VEL
LIN {X 0,Y 588.917,Z 397.344,A -85,B 0,C 180,E1 26588.694,E2 26588.694} C_VEL
LIN {X 0,Y 588.189,Z 603.589,A -85,B 0,C 180,E1 26585.653,E2 26585.653} C_VEL
LIN {X 0,Y 587.71,Z 739.547,A -85,B 0,C 180,E1 26583.677,E2 26583.677} C_VEL
LIN {X 0,Y 587.466,Z 763.238,A -85,B 0,C 180,E1 26583.149,E2 26583.149} C_VEL
LIN {X 0,Y 587.253,Z 783.729,A -85,B 0,C 180,E1 26582.526,E2 26582.526} C_VEL
LIN {X 0,Y 586.874,Z 807.105,A -85,B 0,C 180,E1 26581.619,E2 26581.619} C_VEL
LIN {X 0,Y 586.587,Z 828.561,A -85,B 0,C 180,E1 26580.595,E2 26580.595} C_VEL
LIN {X 0,Y 586.172,Z 849.003,A -85,B 0,C 180,E1 26579.425,E2 26579.425} C_VEL
LIN {X 0,Y 585.845,Z 869.342,A -85,B 0,C 180,E1 26578.072,E2 26578.072} C_VEL
LIN {X 0,Y 585.457,Z 888.557,A -85,B 0,C 180,E1 26576.582,E2 26576.582} C_VEL
LIN {X 0,Y 585.096,Z 907.99,A -85,B 0,C 180,E1 26574.85,E2 26574.85} C_VEL
LIN {X 0,Y 584.849,Z 925.079,A -85,B 0,C 180,E1 26573.109,E2 26573.109} C_VEL
LIN {X 0,Y 584.574,Z 941.126,A -85,B 0,C 180,E1 26571.225,E2 26571.225} C_VEL
LIN {X 0,Y 584.344,Z 956.346,A -85,B 0,C 180,E1 26569.177,E2 26569.177} C_VEL
LIN {X 0,Y 584.206,Z 969.63,A -85,B 0,C 180,E1 26567.122,E2 26567.122} C_VEL
LIN {X 0,Y 584.086,Z 980.823,A -85,B 0,C 180,E1 26565.084,E2 26565.084} C_VEL
LIN {X 0,Y 584.007,Z 990.868,A -85,B 0,C 180,E1 26562.963,E2 26562.963} C_VEL
LIN {X 0,Y 583.937,Z 999.041,A -85,B 0,C 180,E1 26560.859,E2 26560.859} C_VEL
LIN {X 0,Y 583.928,Z 1006.033,A -85,B 0,C 180,E1 26558.669,E2 26558.669} C_VEL
LIN {X 0,Y 583.921,Z 1011.248,A -85,B 0,C 180,E1 26556.492,E2 26556.492} C_VEL
LIN {X 0,Y 583.912,Z 1015.16,A -85,B 0,C 180,E1 26554.225,E2 26554.225} C_VEL
LIN {X 0,Y 583.915,Z 1017.254,A -85,B 0,C 180,E1 26552.064,E2 26552.064} C_VEL
LIN {X 0,Y 583.9,Z 1017.962,A -85,B 0,C 180,E1 26549.807,E2 26549.807} C_VEL
LIN {X 0,Y 583.915,Z 1017.124,A -85,B 0,C 180,E1 26547.746,E2 26547.746} C_VEL
LIN {X 0,Y 583.9,Z 1014.758,A -85,B 0,C 180,E1 26545.485,E2 26545.485} C_VEL
LIN {X 0,Y 583.913,Z 1011.054,A -85,B 0,C 180,E1 26543.415,E2 26543.415} C_VEL
LIN {X 0,Y 583.93,Z 1005.785,A -85,B 0,C 180,E1 26541.238,E2 26541.238} C_VEL
LIN {X 0,Y 583.937,Z 999.062,A -85,B 0,C 180,E1 26539.147,E2 26539.147} C_VEL
LIN {X 0,Y 584.01,Z 990.893,A -85,B 0,C 180,E1 26537.043,E2 26537.043} C_VEL
LIN {X 0,Y 584.088,Z 980.734,A -85,B 0,C 180,E1 26534.898,E2 26534.898} C_VEL
LIN {X 0,Y 584.211,Z 969.037,A -85,B 0,C 180,E1 26532.781,E2 26532.781} C_VEL
LIN {X 0,Y 584.344,Z 956.346,A -85,B 0,C 180,E1 26530.823,E2 26530.823} C_VEL
LIN {X 0,Y 584.573,Z 940.875,A -85,B 0,C 180,E1 26528.744,E2 26528.744} C_VEL
LIN {X 0,Y 584.855,Z 924.713,A -85,B 0,C 180,E1 26526.85,E2 26526.85} C_VEL
LIN {X 0,Y 585.098,Z 907.948,A -85,B 0,C 180,E1 26525.146,E2 26525.146} C_VEL
LIN {X 0,Y 585.456,Z 888.636,A -85,B 0,C 180,E1 26523.424,E2 26523.424} C_VEL
LIN {X 0,Y 585.835,Z 869.665,A -85,B 0,C 180,E1 26521.952,E2 26521.952} C_VEL
LIN {X 0,Y 586.17,Z 849.11,A -85,B 0,C 180,E1 26520.582,E2 26520.582} C_VEL
LIN {X 0,Y 586.594,Z 827.76,A -85,B 0,C 180,E1 26519.364,E2 26519.364} C_VEL
LIN {X 0,Y 586.874,Z 807.182,A -85,B 0,C 180,E1 26518.384,E2 26518.384} C_VEL
LIN {X 0,Y 587.251,Z 783.94,A -85,B 0,C 180,E1 26517.481,E2 26517.481} C_VEL
LIN {X 0,Y 587.465,Z 763.452,A -85,B 0,C 180,E1 26516.857,E2 26516.857} C_VEL
LIN {X 0,Y 587.708,Z 739.75,A -85,B 0,C 180,E1 26516.326,E2 26516.326} C_VEL
LIN {X 0,Y 588.14,Z 616.113,A -85,B 0,C 180,E1 26514.528,E2 26514.528} C_VEL
LIN {X 0,Y 588.88,Z 407.862,A -85,B 0,C 180,E1 26511.464,E2 26511.464} C_VEL
LIN {X 0,Y 588.741,Z 395.52,A -85,B 0,C 180,E1 26511.265,E2 26511.265} C_VEL
LIN {X 0,Y 587.759,Z 390.12,A -85,B 0,C 180,E1 26511.061,E2 26511.061} C_VEL
LIN {X 0,Y 587.942,Z 367.547,A -85,B 0,C 180,E1 26509.479,E2 26509.479} C_VEL
LIN {X 0,Y 584.146,Z 358.602,A -85,B 0,C 180,E1 26508.479,E2 26508.479} C_VEL
LIN {X 0,Y 584.025,Z 358.267,A -85,B 0,C 180,E1 26507.721,E2 26507.721} C_VEL
LIN {X 0,Y 584.051,Z 358.288,A -85,B 0,C 180,E1 26504.855,E2 26504.855} C_VEL
LIN {X 0,Y 584.027,Z 358.296,A -85,B 0,C 180,E1 26501.577,E2 26501.577} C_VEL
LIN {X 0,Y 584.046,Z 358.289,A -85,B 0,C 180,E1 26498.672,E2 26498.672} C_VEL
LIN {X 0,Y 584.021,Z 358.288,A -85,B 0,C 180,E1 26495.429,E2 26495.429} C_VEL
LIN {X 0,Y 584.03,Z 358.295,A -85,B 0,C 180,E1 26492.625,E2 26492.625} C_VEL
LIN {X 0,Y 584.021,Z 358.293,A -85,B 0,C 180,E1 26489.316,E2 26489.316} C_VEL
LIN {X 0,Y 584.018,Z 358.295,A -85,B 0,C 180,E1 26486.541,E2 26486.541} C_VEL
LIN {X 0,Y 584.023,Z 358.294,A -85,B 0,C 180,E1 26483.181,E2 26483.181} C_VEL
LIN {X 0,Y 584.023,Z 358.294,A -85,B 0,C 180,E1 26480.336,E2 26480.336} C_VEL
LIN {X 0,Y 584.029,Z 358.294,A -85,B 0,C 180,E1 26477.022,E2 26477.022} C_VEL
LIN {X 0,Y 584.026,Z 358.293,A -85,B 0,C 180,E1 26474.171,E2 26474.171} C_VEL
LIN {X 0,Y 584.034,Z 358.293,A -85,B 0,C 180,E1 26470.854,E2 26470.854} C_VEL
LIN {X 0,Y 584.033,Z 358.292,A -85,B 0,C 180,E1 26467.971,E2 26467.971} C_VEL
LIN {X 0,Y 584.035,Z 358.292,A -85,B 0,C 180,E1 26464.615,E2 26464.615} C_VEL
